LIN {X 0,Y 404.133,Z 474.142,A -85,B 0,C 180,E1 -11048.582,E2 -11048.582} C_VEL
LIN {X 0,Y 404.205,Z 474.132,A -85,B 0,C 180,E1 -11051.764,E2 -11051.764} C_VEL
LIN {X 0,Y 404.201,Z 474.136,A -85,B 0,C 180,E1 -11054.884,E2 -11054.884} C_VEL
LIN {X 0,Y 404.253,Z 474.125,A -85,B 0,C 180,E1 -11057.96,E2 -11057.96} C_VEL
LIN {X 0,Y 404.43,Z 474.108,A -85,B 0,C 180,E1 -11062.101,E2 -11062.101} C_VEL
LIN {X 0,Y 404.423,Z 474.111,A -85,B 0,C 180,E1 -11064.017,E2 -11064.017} C_VEL
LIN {X 0,Y 404.303,Z 474.258,A -85,B 0,C 180,E1 -11065.079,E2 -11065.079} C_VEL
LIN {X 0,Y 404.496,Z 475.213,A -85,B 0,C 180,E1 -11065.255,E2 -11065.255} C_VEL
LIN {X 0,Y 409.813,Z 489.68,A -85,B 0,C 180,E1 -11065.753,E2 -11065.753} C_VEL
LIN {X 0,Y 409.191,Z 554.574,A -85,B 0,C 180,E1 -11066.911,E2 -11066.911} C_VEL
LIN {X 0,Y 409.132,Z 567.718,A -85,B 0,C 180,E1 -11067.325,E2 -11067.325} C_VEL
LIN {X 0,Y 408.856,Z 581.109,A -85,B 0,C 180,E1 -11067.97,E2 -11067.97} C_VEL
LIN {X 0,Y 408.461,Z 593.219,A -85,B 0,C 180,E1 -11068.769,E2 -11068.769} C_VEL
LIN {X 0,Y 407.969,Z 603.324,A -85,B 0,C 180,E1 -11069.625,E2 -11069.625} C_VEL
LIN {X 0,Y 407.316,Z 613.938,A -85,B 0,C 180,E1 -11070.743,E2 -11070.743} C_VEL
LIN {X 0,Y 406.77,Z 623.415,A -85,B 0,C 180,E1 -11071.982,E2 -11071.982} C_VEL
LIN {X 0,Y 406.186,Z 631.224,A -85,B 0,C 180,E1 -11073.225,E2 -11073.225} C_VEL
LIN {X 0,Y 405.837,Z 635.869,A -85,B 0,C 180,E1 -11074.098,E2 -11074.098} C_VEL
LIN {X 0,Y 404.918,Z 639.248,A -85,B 0,C 180,E1 -11074.777,E2 -11074.777} C_VEL
LIN {X 0,Y 401.737,Z 644.43,A -85,B 0,C 180,E1 -11075.892,E2 -11075.892} C_VEL
LIN {X 0,Y 398.611,Z 648.964,A -85,B 0,C 180,E1 -11077.072,E2 -11077.072} C_VEL
LIN {X 0,Y 397.791,Z 651.292,A -85,B 0,C 180,E1 -11077.842,E2 -11077.842} C_VEL
LIN {X 0,Y 397.533,Z 654.48,A -85,B 0,C 180,E1 -11079.157,E2 -11079.157} C_VEL
LIN {X 0,Y 397.346,Z 656.459,A -85,B 0,C 180,E1 -11080.189,E2 -11080.189} C_VEL
LIN {X 0,Y 397.231,Z 658.018,A -85,B 0,C 180,E1 -11081.224,E2 -11081.224} C_VEL
LIN {X 0,Y 397.183,Z 659.113,A -85,B 0,C 180,E1 -11082.261,E2 -11082.261} C_VEL
LIN {X 0,Y 397.191,Z 659.81,A -85,B 0,C 180,E1 -11083.3,E2 -11083.3} C_VEL
LIN {X 0,Y 397.189,Z 660.13,A -85,B 0,C 180,E1 -11084.344,E2 -11084.344} C_VEL
LIN {X 0,Y 397.243,Z 660.03,A -85,B 0,C 180,E1 -11085.391,E2 -11085.391} C_VEL
LIN {X 0,Y 397.477,Z 658.759,A -85,B 0,C 180,E1 -11087.293,E2 -11087.293} C_VEL
LIN {X 0,Y 397.711,Z 657.198,A -85,B 0,C 180,E1 -11088.548,E2 -11088.548} C_VEL
LIN {X 0,Y 398.123,Z 654.276,A -85,B 0,C 180,E1 -11090.136,E2 -11090.136} C_VEL
LIN {X 0,Y 398.652,Z 650.226,A -85,B 0,C 180,E1 -11091.731,E2 -11091.731} C_VEL
LIN {X 0,Y 399.254,Z 644.972,A -85,B 0,C 180,E1 -11093.315,E2 -11093.315} C_VEL
LIN {X 0,Y 400.042,Z 638.106,A -85,B 0,C 180,E1 -11094.939,E2 -11094.939} C_VEL
LIN {X 0,Y 400.989,Z 629.888,A -85,B 0,C 180,E1 -11096.484,E2 -11096.484} C_VEL
LIN {X 0,Y 401.872,Z 620.477,A -85,B 0,C 180,E1 -11097.894,E2 -11097.894} C_VEL
LIN {X 0,Y 402.692,Z 610.549,A -85,B 0,C 180,E1 -11099.095,E2 -11099.095} C_VEL
LIN {X 0,Y 403.461,Z 600.695,A -85,B 0,C 180,E1 -11100.055,E2 -11100.055} C_VEL
LIN {X 0,Y 404.094,Z 589.275,A -85,B 0,C 180,E1 -11100.942,E2 -11100.942} C_VEL
LIN {X 0,Y 404.526,Z 577.358,A -85,B 0,C 180,E1 -11101.648,E2 -11101.648} C_VEL
LIN {X 0,Y 404.762,Z 564.049,A -85,B 0,C 180,E1 -11102.21,E2 -11102.21} C_VEL
LIN {X 0,Y 404.819,Z 549.962,A -85,B 0,C 180,E1 -11102.562,E2 -11102.562} C_VEL
LIN {X 0,Y 405.482,Z 494.287,A -85,B 0,C 180,E1 -11103.583,E2 -11103.583} C_VEL
LIN {X 0,Y 397.314,Z 475.91,A -85,B 0,C 180,E1 -11104.495,E2 -11104.495} C_VEL
LIN {X 0,Y 397.145,Z 475.073,A -85,B 0,C 180,E1 -11104.724,E2 -11104.724} C_VEL
LIN {X 0,Y 397.104,Z 475.022,A -85,B 0,C 180,E1 -11108.277,E2 -11108.277} C_VEL
LIN {X 0,Y 397.093,Z 475.024,A -85,B 0,C 180,E1 -11110.91,E2 -11110.91} C_VEL
LIN {X 0,Y 397.105,Z 475.019,A -85,B 0,C 180,E1 -11113.65,E2 -11113.65} C_VEL
LIN {X 0,Y 397.107,Z 475.021,A -85,B 0,C 180,E1 -11116.522,E2 -11116.522} C_VEL
LIN {X 0,Y 397.133,Z 475.196,A -85,B 0,C 180,E1 -11119.013,E2 -11119.013} C_VEL
LIN {X 0,Y 399.935,Z 487.895,A -85,B 0,C 180,E1 -11121.445,E2 -11121.445} C_VEL
LIN {X 0,Y 401.126,Z 495.291,A -85,B 0,C 180,E1 -11122.81,E2 -11122.81} C_VEL
LIN {X 0,Y 400.2,Z 516.124,A -85,B 0,C 180,E1 -11126.415,E2 -11126.415} C_VEL
LIN {X 0,Y 399.995,Z 522.02,A -85,B 0,C 180,E1 -11127.397,E2 -11127.397} C_VEL
LIN {X 0,Y 403.104,Z 541.761,A -85,B 0,C 180,E1 -11127.979,E2 -11127.979} C_VEL
LIN {X 0,Y 401.336,Z 632.644,A -85,B 0,C 180,E1 -11129.88,E2 -11129.88} C_VEL
LIN {X 0,Y 401.005,Z 645.03,A -85,B 0,C 180,E1 -11130.324,E2 -11130.324} C_VEL
LIN {X 0,Y 400.448,Z 657.146,A -85,B 0,C 180,E1 -11130.945,E2 -11130.945} C_VEL
LIN {X 0,Y 399.891,Z 669.821,A -85,B 0,C 180,E1 -11131.815,E2 -11131.815} C_VEL
LIN {X 0,Y 399.221,Z 680.557,A -85,B 0,C 180,E1 -11132.761,E2 -11132.761} C_VEL
LIN {X 0,Y 398.431,Z 692.076,A -85,B 0,C 180,E1 -11134.034,E2 -11134.034} C_VEL
LIN {X 0,Y 397.889,Z 700.606,A -85,B 0,C 180,E1 -11135.197,E2 -11135.197} C_VEL
LIN {X 0,Y 397.334,Z 708.675,A -85,B 0,C 180,E1 -11136.534,E2 -11136.534} C_VEL
LIN {X 0,Y 396.781,Z 716.618,A -85,B 0,C 180,E1 -11138.164,E2 -11138.164} C_VEL
LIN {X 0,Y 396.441,Z 722.686,A -85,B 0,C 180,E1 -11139.733,E2 -11139.733} C_VEL
LIN {X 0,Y 396.136,Z 727.578,A -85,B 0,C 180,E1 -11141.377,E2 -11141.377} C_VEL
LIN {X 0,Y 396.042,Z 730.058,A -85,B 0,C 180,E1 -11142.442,E2 -11142.442} C_VEL
LIN {X 0,Y 395.913,Z 732.043,A -85,B 0,C 180,E1 -11143.5,E2 -11143.5} C_VEL
LIN {X 0,Y 395.806,Z 733.503,A -85,B 0,C 180,E1 -11144.554,E2 -11144.554} C_VEL
LIN {X 0,Y 395.753,Z 734.538,A -85,B 0,C 180,E1 -11145.605,E2 -11145.605} C_VEL
LIN {X 0,Y 395.865,Z 735.231,A -85,B 0,C 180,E1 -11147.544,E2 -11147.544} C_VEL
LIN {X 0,Y 395.892,Z 734.913,A -85,B 0,C 180,E1 -11148.74,E2 -11148.74} C_VEL
LIN {X 0,Y 395.902,Z 734.17,A -85,B 0,C 180,E1 -11149.775,E2 -11149.775} C_VEL
LIN {X 0,Y 396.034,Z 732.96,A -85,B 0,C 180,E1 -11150.81,E2 -11150.81} C_VEL
LIN {X 0,Y 396.277,Z 730.336,A -85,B 0,C 180,E1 -11152.357,E2 -11152.357} C_VEL
LIN {X 0,Y 396.521,Z 726.682,A -85,B 0,C 180,E1 -11153.896,E2 -11153.896} C_VEL
LIN {X 0,Y 396.894,Z 721.882,A -85,B 0,C 180,E1 -11155.43,E2 -11155.43} C_VEL
LIN {X 0,Y 397.41,Z 715.803,A -85,B 0,C 180,E1 -11156.959,E2 -11156.959} C_VEL
LIN {X 0,Y 398.122,Z 708.162,A -85,B 0,C 180,E1 -11158.483,E2 -11158.483} C_VEL
LIN {X 0,Y 399.009,Z 698.649,A -85,B 0,C 180,E1 -11160,E2 -11160} C_VEL
LIN {X 0,Y 399.831,Z 688.759,A -85,B 0,C 180,E1 -11161.259,E2 -11161.259} C_VEL
LIN {X 0,Y 400.716,Z 677.71,A -85,B 0,C 180,E1 -11162.388,E2 -11162.388} C_VEL
LIN {X 0,Y 401.413,Z 666.543,A -85,B 0,C 180,E1 -11163.301,E2 -11163.301} C_VEL
LIN {X 0,Y 402.197,Z 653.515,A -85,B 0,C 180,E1 -11164.108,E2 -11164.108} C_VEL
LIN {X 0,Y 402.666,Z 640.568,A -85,B 0,C 180,E1 -11164.692,E2 -11164.692} C_VEL
LIN {X 0,Y 403.089,Z 626.256,A -85,B 0,C 180,E1 -11165.096,E2 -11165.096} C_VEL
LIN {X 0,Y 405.254,Z 541.083,A -85,B 0,C 180,E1 -11166.99,E2 -11166.99} C_VEL
LIN {X 0,Y 402.058,Z 526.063,A -85,B 0,C 180,E1 -11167.597,E2 -11167.597} C_VEL
LIN {X 0,Y 401.812,Z 524.403,A -85,B 0,C 180,E1 -11167.728,E2 -11167.728} C_VEL
LIN {X 0,Y 402.819,Z 502.886,A -85,B 0,C 180,E1 -11171.411,E2 -11171.411} C_VEL
LIN {X 0,Y 403.071,Z 499.016,A -85,B 0,C 180,E1 -11172.078,E2 -11172.078} C_VEL
LIN {X 0,Y 401.479,Z 490.655,A -85,B 0,C 180,E1 -11173.67,E2 -11173.67} C_VEL
LIN {X 0,Y 398.591,Z 479.718,A -85,B 0,C 180,E1 -11175.861,E2 -11175.861} C_VEL
LIN {X 0,Y 397.195,Z 475.127,A -85,B 0,C 180,E1 -11176.877,E2 -11176.877} C_VEL
LIN {X 0,Y 397.148,Z 475.016,A -85,B 0,C 180,E1 -11180.295,E2 -11180.295} C_VEL
LIN {X 0,Y 397.134,Z 475.017,A -85,B 0,C 180,E1 -11184.019,E2 -11184.019} C_VEL
LIN {X 0,Y 397.203,Z 475.009,A -85,B 0,C 180,E1 -11187.39,E2 -11187.39} C_VEL
LIN {X 0,Y 397.088,Z 475.024,A -85,B 0,C 180,E1 -11190.882,E2 -11190.882} C_VEL
LIN {X 0,Y 397.134,Z 475.016,A -85,B 0,C 180,E1 -11194.493,E2 -11194.493} C_VEL
LIN {X 0,Y 397.11,Z 475.017,A -85,B 0,C 180,E1 -11198.275,E2 -11198.275} C_VEL
LIN {X 0,Y 397.097,Z 475.023,A -85,B 0,C 180,E1 -11200.908,E2 -11200.908} C_VEL
LIN {X 0,Y 397.109,Z 475.019,A -85,B 0,C 180,E1 -11203.648,E2 -11203.648} C_VEL
LIN {X 0,Y 397.11,Z 475.018,A -85,B 0,C 180,E1 -11206.52,E2 -11206.52} C_VEL
LIN {X 0,Y 397.12,Z 475.008,A -85,B 0,C 180,E1 -11210.422,E2 -11210.422} C_VEL
LIN {X 0,Y 397.104,Z 475.007,A -85,B 0,C 180,E1 -11213.004,E2 -11213.004} C_VEL
LIN {X 0,Y 397.146,Z 475.218,A -85,B 0,C 180,E1 -11215.91,E2 -11215.91} C_VEL
LIN {X 0,Y 400.382,Z 487.87,A -85,B 0,C 180,E1 -11218.488,E2 -11218.488} C_VEL
LIN {X 0,Y 402.986,Z 499.886,A -85,B 0,C 180,E1 -11220.769,E2 -11220.769} C_VEL
LIN {X 0,Y 402.926,Z 503.223,A -85,B 0,C 180,E1 -11221.335,E2 -11221.335} C_VEL
LIN {X 0,Y 401.063,Z 524.8,A -85,B 0,C 180,E1 -11224.851,E2 -11224.851} C_VEL
LIN {X 0,Y 399.235,Z 550.114,A -85,B 0,C 180,E1 -11228.907,E2 -11228.907} C_VEL
LIN {X 0,Y 399.204,Z 552.057,A -85,B 0,C 180,E1 -11229.132,E2 -11229.132} C_VEL
LIN {X 0,Y 400.616,Z 562.417,A -85,B 0,C 180,E1 -11229.554,E2 -11229.554} C_VEL
LIN {X 0,Y 403.001,Z 585.438,A -85,B 0,C 180,E1 -11230.266,E2 -11230.266} C_VEL
LIN {X 0,Y 403.893,Z 597.547,A -85,B 0,C 180,E1 -11230.544,E2 -11230.544} C_VEL
LIN {X 0,Y 402.92,Z 664.118,A -85,B 0,C 180,E1 -11231.766,E2 -11231.766} C_VEL
LIN {X 0,Y 402.288,Z 677.425,A -85,B 0,C 180,E1 -11232.197,E2 -11232.197} C_VEL
LIN {X 0,Y 401.369,Z 690.214,A -85,B 0,C 180,E1 -11232.812,E2 -11232.812} C_VEL
LIN {X 0,Y 399.991,Z 709.915,A -85,B 0,C 180,E1 -11234.064,E2 -11234.064} C_VEL
LIN {X 0,Y 399.197,Z 720.793,A -85,B 0,C 180,E1 -11234.947,E2 -11234.947} C_VEL
LIN {X 0,Y 398.466,Z 730.713,A -85,B 0,C 180,E1 -11235.948,E2 -11235.948} C_VEL
LIN {X 0,Y 397.619,Z 741.025,A -85,B 0,C 180,E1 -11237.234,E2 -11237.234} C_VEL
LIN {X 0,Y 397.105,Z 749.384,A -85,B 0,C 180,E1 -11238.514,E2 -11238.514} C_VEL
LIN {X 0,Y 396.569,Z 757.583,A -85,B 0,C 180,E1 -11240.048,E2 -11240.048} C_VEL
LIN {X 0,Y 396.182,Z 765.089,A -85,B 0,C 180,E1 -11241.84,E2 -11241.84} C_VEL
LIN {X 0,Y 395.994,Z 770.249,A -85,B 0,C 180,E1 -11243.425,E2 -11243.425} C_VEL
LIN {X 0,Y 395.987,Z 773.916,A -85,B 0,C 180,E1 -11244.907,E2 -11244.907} C_VEL
LIN {X 0,Y 395.92,Z 775.85,A -85,B 0,C 180,E1 -11245.927,E2 -11245.927} C_VEL
LIN {X 0,Y 395.972,Z 777.314,A -85,B 0,C 180,E1 -11246.946,E2 -11246.946} C_VEL
LIN {X 0,Y 396.014,Z 778.36,A -85,B 0,C 180,E1 -11247.964,E2 -11247.964} C_VEL
LIN {X 0,Y 395.992,Z 778.965,A -85,B 0,C 180,E1 -11248.981,E2 -11248.981} C_VEL
LIN {X 0,Y 396.085,Z 779.104,A -85,B 0,C 180,E1 -11249.998,E2 -11249.998} C_VEL
LIN {X 0,Y 396.014,Z 778.816,A -85,B 0,C 180,E1 -11251.015,E2 -11251.015} C_VEL
LIN {X 0,Y 396.013,Z 778.114,A -85,B 0,C 180,E1 -11252.032,E2 -11252.032} C_VEL
LIN {X 0,Y 396.018,Z 776.927,A -85,B 0,C 180,E1 -11253.05,E2 -11253.05} C_VEL
LIN {X 0,Y 395.971,Z 774.309,A -85,B 0,C 180,E1 -11254.579,E2 -11254.579} C_VEL
LIN {X 0,Y 395.971,Z 770.015,A -85,B 0,C 180,E1 -11256.313,E2 -11256.313} C_VEL
LIN {X 0,Y 396.099,Z 765.675,A -85,B 0,C 180,E1 -11257.645,E2 -11257.645} C_VEL
LIN {X 0,Y 396.328,Z 759.409,A -85,B 0,C 180,E1 -11259.182,E2 -11259.182} C_VEL
LIN {X 0,Y 396.698,Z 751.537,A -85,B 0,C 180,E1 -11260.719,E2 -11260.719} C_VEL
LIN {X 0,Y 397.179,Z 743.415,A -85,B 0,C 180,E1 -11261.998,E2 -11261.998} C_VEL
LIN {X 0,Y 397.828,Z 734.585,A -85,B 0,C 180,E1 -11263.145,E2 -11263.145} C_VEL
LIN {X 0,Y 398.362,Z 723.74,A -85,B 0,C 180,E1 -11264.298,E2 -11264.298} C_VEL
LIN {X 0,Y 399.039,Z 713.221,A -85,B 0,C 180,E1 -11265.186,E2 -11265.186} C_VEL
LIN {X 0,Y 399.761,Z 700.61,A -85,B 0,C 180,E1 -11266.007,E2 -11266.007} C_VEL
LIN {X 0,Y 400.839,Z 683.335,A -85,B 0,C 180,E1 -11266.945,E2 -11266.945} C_VEL
LIN {X 0,Y 401.414,Z 670.298,A -85,B 0,C 180,E1 -11267.445,E2 -11267.445} C_VEL
LIN {X 0,Y 401.724,Z 654.557,A -85,B 0,C 180,E1 -11267.793,E2 -11267.793} C_VEL
LIN {X 0,Y 402.305,Z 593.458,A -85,B 0,C 180,E1 -11268.885,E2 -11268.885} C_VEL
LIN {X 0,Y 398.442,Z 555.652,A -85,B 0,C 180,E1 -11269.746,E2 -11269.746} C_VEL
LIN {X 0,Y 398.417,Z 554.31,A -85,B 0,C 180,E1 -11269.848,E2 -11269.848} C_VEL
LIN {X 0,Y 399.688,Z 532.021,A -85,B 0,C 180,E1 -11273.303,E2 -11273.303} C_VEL
LIN {X 0,Y 401.324,Z 507.919,A -85,B 0,C 180,E1 -11277.083,E2 -11277.083} C_VEL
LIN {X 0,Y 401.936,Z 497.094,A -85,B 0,C 180,E1 -11278.805,E2 -11278.805} C_VEL
LIN {X 0,Y 397.969,Z 478.817,A -85,B 0,C 180,E1 -11282.041,E2 -11282.041} C_VEL
LIN {X 0,Y 397.143,Z 475.144,A -85,B 0,C 180,E1 -11282.738,E2 -11282.738} C_VEL
LIN {X 0,Y 397.1,Z 475.022,A -85,B 0,C 180,E1 -11285.733,E2 -11285.733} C_VEL
LIN {X 0,Y 397.084,Z 475.019,A -85,B 0,C 180,E1 -11288.852,E2 -11288.852} C_VEL
LIN {X 0,Y 397.048,Z 475.029,A -85,B 0,C 180,E1 -11292.267,E2 -11292.267} C_VEL
LIN {X 0,Y 397.077,Z 475.019,A -85,B 0,C 180,E1 -11295.067,E2 -11295.067} C_VEL
LIN {X 0,Y 397.05,Z 475.027,A -85,B 0,C 180,E1 -11298.021,E2 -11298.021} C_VEL
LIN {X 0,Y 397.084,Z 475.018,A -85,B 0,C 180,E1 -11301.144,E2 -11301.144} C_VEL
LIN {X 0,Y 397.108,Z 475.02,A -85,B 0,C 180,E1 -11304.495,E2 -11304.495} C_VEL
LIN {X 0,Y 397.067,Z 475.023,A -85,B 0,C 180,E1 -11307.927,E2 -11307.927} C_VEL
LIN {X 0,Y 397.11,Z 475.015,A -85,B 0,C 180,E1 -11311.455,E2 -11311.455} C_VEL
LIN {X 0,Y 397.139,Z 475.017,A -85,B 0,C 180,E1 -11314.487,E2 -11314.487} C_VEL
LIN {X 0,Y 397.096,Z 475.022,A -85,B 0,C 180,E1 -11318.181,E2 -11318.181} C_VEL
LIN {X 0,Y 397.149,Z 475.01,A -85,B 0,C 180,E1 -11321.426,E2 -11321.426} C_VEL
LIN {X 0,Y 397.165,Z 475.013,A -85,B 0,C 180,E1 -11324.607,E2 -11324.607} C_VEL
LIN {X 0,Y 397.207,Z 475.004,A -85,B 0,C 180,E1 -11327.741,E2 -11327.741} C_VEL
LIN {X 0,Y 397.381,Z 474.984,A -85,B 0,C 180,E1 -11332.041,E2 -11332.041} C_VEL
LIN {X 0,Y 397.238,Z 475.002,A -85,B 0,C 180,E1 -11334.925,E2 -11334.925} C_VEL
LIN {X 0,Y 397.435,Z 474.976,A -85,B 0,C 180,E1 -11337.973,E2 -11337.973} C_VEL
LIN {X 0,Y 397.566,Z 474.96,A -85,B 0,C 180,E1 -11340,E2 -11340} C_VEL
LIN {X 0,Y 397.366,Z 474.985,A -85,B 0,C 180,E1 -11343.041,E2 -11343.041} C_VEL
LIN {X 0,Y 397.348,Z 474.987,A -85,B 0,C 180,E1 -11347.112,E2 -11347.112} C_VEL
LIN {X 0,Y 397.205,Z 475.006,A -85,B 0,C 180,E1 -11350.191,E2 -11350.191} C_VEL
LIN {X 0,Y 397.212,Z 475.003,A -85,B 0,C 180,E1 -11353.321,E2 -11353.321} C_VEL
LIN {X 0,Y 397.167,Z 475.01,A -85,B 0,C 180,E1 -11357.155,E2 -11357.155} C_VEL
LIN {X 0,Y 397.088,Z 475.025,A -85,B 0,C 180,E1 -11360.73,E2 -11360.73} C_VEL
LIN {X 0,Y 397.119,Z 475.014,A -85,B 0,C 180,E1 -11364.019,E2 -11364.019} C_VEL
LIN {X 0,Y 397.181,Z 475.007,A -85,B 0,C 180,E1 -11367.391,E2 -11367.391} C_VEL
LIN {X 0,Y 397.066,Z 475.027,A -85,B 0,C 180,E1 -11370.883,E2 -11370.883} C_VEL
LIN {X 0,Y 397.113,Z 475.018,A -85,B 0,C 180,E1 -11374.494,E2 -11374.494} C_VEL
LIN {X 0,Y 397.092,Z 475.019,A -85,B 0,C 180,E1 -11378.276,E2 -11378.276} C_VEL
LIN {X 0,Y 397.077,Z 475.026,A -85,B 0,C 180,E1 -11380.91,E2 -11380.91} C_VEL
LIN {X 0,Y 397.094,Z 475.017,A -85,B 0,C 180,E1 -11383.649,E2 -11383.649} C_VEL
LIN {X 0,Y 397.149,Z 475.013,A -85,B 0,C 180,E1 -11386.513,E2 -11386.513} C_VEL
LIN {X 0,Y 397.114,Z 475.016,A -85,B 0,C 180,E1 -11389.552,E2 -11389.552} C_VEL
LIN {X 0,Y 397.113,Z 475.02,A -85,B 0,C 180,E1 -11392.787,E2 -11392.787} C_VEL
LIN {X 0,Y 397.109,Z 475.016,A -85,B 0,C 180,E1 -11396.284,E2 -11396.284} C_VEL
LIN {X 0,Y 397.097,Z 475.017,A -85,B 0,C 180,E1 -11400.137,E2 -11400.137} C_VEL
LIN {X 0,Y 397.187,Z 475.008,A -85,B 0,C 180,E1 -11402.611,E2 -11402.611} C_VEL
LIN {X 0,Y 397.126,Z 475.013,A -85,B 0,C 180,E1 -11405.983,E2 -11405.983} C_VEL
LIN {X 0,Y 397.132,Z 475.013,A -85,B 0,C 180,E1 -11409.706,E2 -11409.706} C_VEL
LIN {X 0,Y 397.176,Z 475.011,A -85,B 0,C 180,E1 -11412.846,E2 -11412.846} C_VEL
LIN {X 0,Y 397.224,Z 475.003,A -85,B 0,C 180,E1 -11416.704,E2 -11416.704} C_VEL
LIN {X 0,Y 397.215,Z 475.007,A -85,B 0,C 180,E1 -11419.811,E2 -11419.811} C_VEL
LIN {X 0,Y 397.362,Z 474.988,A -85,B 0,C 180,E1 -11422.89,E2 -11422.89} C_VEL
LIN {X 0,Y 397.274,Z 475.174,A -85,B 0,C 180,E1 -11424.8,E2 -11424.8} C_VEL
LIN {X 0,Y 397.434,Z 476.035,A -85,B 0,C 180,E1 -11424.957,E2 -11424.957} C_VEL
LIN {X 0,Y 402.904,Z 491.025,A -85,B 0,C 180,E1 -11425.492,E2 -11425.492} C_VEL
LIN {X 0,Y 402.371,Z 556.242,A -85,B 0,C 180,E1 -11426.68,E2 -11426.68} C_VEL
LIN {X 0,Y 402.262,Z 569.599,A -85,B 0,C 180,E1 -11427.123,E2 -11427.123} C_VEL
LIN {X 0,Y 401.992,Z 582.198,A -85,B 0,C 180,E1 -11427.747,E2 -11427.747} C_VEL
LIN {X 0,Y 401.614,Z 593.455,A -85,B 0,C 180,E1 -11428.498,E2 -11428.498} C_VEL
LIN {X 0,Y 401.072,Z 604.477,A -85,B 0,C 180,E1 -11429.442,E2 -11429.442} C_VEL
LIN {X 0,Y 400.362,Z 615.489,A -85,B 0,C 180,E1 -11430.63,E2 -11430.63} C_VEL
LIN {X 0,Y 399.883,Z 623.984,A -85,B 0,C 180,E1 -11431.764,E2 -11431.764} C_VEL
LIN {X 0,Y 399.269,Z 631.862,A -85,B 0,C 180,E1 -11433.029,E2 -11433.029} C_VEL
LIN {X 0,Y 398.681,Z 639.577,A -85,B 0,C 180,E1 -11434.552,E2 -11434.552} C_VEL
LIN {X 0,Y 398.214,Z 645.749,A -85,B 0,C 180,E1 -11436.08,E2 -11436.08} C_VEL
LIN {X 0,Y 397.791,Z 651.292,A -85,B 0,C 180,E1 -11437.842,E2 -11437.842} C_VEL
LIN {X 0,Y 396.97,Z 653.417,A -85,B 0,C 180,E1 -11438.629,E2 -11438.629} C_VEL
LIN {X 0,Y 393.875,Z 656.494,A -85,B 0,C 180,E1 -11439.919,E2 -11439.919} C_VEL
LIN {X 0,Y 391.324,Z 658.509,A -85,B 0,C 180,E1 -11440.982,E2 -11440.982} C_VEL
LIN {X 0,Y 390.234,Z 659.652,A -85,B 0,C 180,E1 -11441.819,E2 -11441.819} C_VEL
LIN {X 0,Y 390.147,Z 659.892,A -85,B 0,C 180,E1 -11442.105,E2 -11442.105} C_VEL
LIN {X 0,Y 390.166,Z 660.9,A -85,B 0,C 180,E1 -11443.544,E2 -11443.544} C_VEL
LIN {X 0,Y 390.166,Z 661.14,A -85,B 0,C 180,E1 -11444.608,E2 -11444.608} C_VEL
LIN {X 0,Y 390.253,Z 660.934,A -85,B 0,C 180,E1 -11445.674,E2 -11445.674} C_VEL
LIN {X 0,Y 390.487,Z 659.688,A -85,B 0,C 180,E1 -11447.467,E2 -11447.467} C_VEL
LIN {X 0,Y 390.768,Z 657.858,A -85,B 0,C 180,E1 -11448.89,E2 -11448.89} C_VEL
LIN {X 0,Y 391.222,Z 654.876,A -85,B 0,C 180,E1 -11450.474,E2 -11450.474} C_VEL
LIN {X 0,Y 391.827,Z 650.601,A -85,B 0,C 180,E1 -11452.129,E2 -11452.129} C_VEL
LIN {X 0,Y 392.46,Z 645.466,A -85,B 0,C 180,E1 -11453.668,E2 -11453.668} C_VEL
LIN {X 0,Y 393.381,Z 638.154,A -85,B 0,C 180,E1 -11455.391,E2 -11455.391} C_VEL
LIN {X 0,Y 394.256,Z 630.587,A -85,B 0,C 180,E1 -11456.809,E2 -11456.809} C_VEL
LIN {X 0,Y 395.212,Z 620.96,A -85,B 0,C 180,E1 -11458.261,E2 -11458.261} C_VEL
LIN {X 0,Y 396.059,Z 611.137,A -85,B 0,C 180,E1 -11459.458,E2 -11459.458} C_VEL
LIN {X 0,Y 396.907,Z 600.915,A -85,B 0,C 180,E1 -11460.457,E2 -11460.457} C_VEL
LIN {X 0,Y 397.578,Z 589.209,A -85,B 0,C 180,E1 -11461.359,E2 -11461.359} C_VEL
LIN {X 0,Y 398.043,Z 576.36,A -85,B 0,C 180,E1 -11462.107,E2 -11462.107} C_VEL
LIN {X 0,Y 398.233,Z 564.269,A -85,B 0,C 180,E1 -11462.604,E2 -11462.604} C_VEL
LIN {X 0,Y 398.269,Z 549.837,A -85,B 0,C 180,E1 -11462.958,E2 -11462.958} C_VEL
LIN {X 0,Y 399.017,Z 496.122,A -85,B 0,C 180,E1 -11463.956,E2 -11463.956} C_VEL
LIN {X 0,Y 390.342,Z 476.97,A -85,B 0,C 180,E1 -11464.937,E2 -11464.937} C_VEL
LIN {X 0,Y 390.134,Z 476.02,A -85,B 0,C 180,E1 -11465.134,E2 -11465.134} C_VEL
LIN {X 0,Y 390.071,Z 475.89,A -85,B 0,C 180,E1 -11469.219,E2 -11469.219} C_VEL
LIN {X 0,Y 390.046,Z 475.892,A -85,B 0,C 180,E1 -11472.375,E2 -11472.375} C_VEL
LIN {X 0,Y 390.049,Z 475.901,A -85,B 0,C 180,E1 -11475.356,E2 -11475.356} C_VEL
LIN {X 0,Y 390.104,Z 476.111,A -85,B 0,C 180,E1 -11478.743,E2 -11478.743} C_VEL
LIN {X 0,Y 393.147,Z 490.003,A -85,B 0,C 180,E1 -11481.429,E2 -11481.429} C_VEL
LIN {X 0,Y 394.23,Z 496.767,A -85,B 0,C 180,E1 -11482.691,E2 -11482.691} C_VEL
LIN {X 0,Y 393.279,Z 517.823,A -85,B 0,C 180,E1 -11486.36,E2 -11486.36} C_VEL
LIN {X 0,Y 393.127,Z 522.4,A -85,B 0,C 180,E1 -11487.112,E2 -11487.112} C_VEL
LIN {X 0,Y 396.267,Z 542.631,A -85,B 0,C 180,E1 -11487.716,E2 -11487.716} C_VEL
LIN {X 0,Y 394.465,Z 632.37,A -85,B 0,C 180,E1 -11489.633,E2 -11489.633} C_VEL
LIN {X 0,Y 394.077,Z 645.723,A -85,B 0,C 180,E1 -11490.117,E2 -11490.117} C_VEL
LIN {X 0,Y 393.495,Z 658.628,A -85,B 0,C 180,E1 -11490.804,E2 -11490.804} C_VEL
LIN {X 0,Y 392.882,Z 671.217,A -85,B 0,C 180,E1 -11491.704,E2 -11491.704} C_VEL
LIN {X 0,Y 392.096,Z 683.083,A -85,B 0,C 180,E1 -11492.802,E2 -11492.802} C_VEL
LIN {X 0,Y 391.45,Z 692.306,A -85,B 0,C 180,E1 -11493.859,E2 -11493.859} C_VEL
LIN {X 0,Y 390.899,Z 700.635,A -85,B 0,C 180,E1 -11495.007,E2 -11495.007} C_VEL
LIN {X 0,Y 390.311,Z 708.872,A -85,B 0,C 180,E1 -11496.382,E2 -11496.382} C_VEL
LIN {X 0,Y 389.743,Z 716.8,A -85,B 0,C 180,E1 -11498.027,E2 -11498.027} C_VEL
LIN {X 0,Y 389.418,Z 722.111,A -85,B 0,C 180,E1 -11499.396,E2 -11499.396} C_VEL
LIN {X 0,Y 389.119,Z 727.167,A -85,B 0,C 180,E1 -11501.029,E2 -11501.029} C_VEL
LIN {X 0,Y 388.928,Z 730.941,A -85,B 0,C 180,E1 -11502.653,E2 -11502.653} C_VEL
LIN {X 0,Y 388.746,Z 733.557,A -85,B 0,C 180,E1 -11504.266,E2 -11504.266} C_VEL
LIN {X 0,Y 388.666,Z 734.691,A -85,B 0,C 180,E1 -11505.336,E2 -11505.336} C_VEL
LIN {X 0,Y 388.681,Z 735.399,A -85,B 0,C 180,E1 -11506.405,E2 -11506.405} C_VEL
LIN {X 0,Y 388.777,Z 735.659,A -85,B 0,C 180,E1 -11507.472,E2 -11507.472} C_VEL
LIN {X 0,Y 388.798,Z 735.452,A -85,B 0,C 180,E1 -11508.531,E2 -11508.531} C_VEL
LIN {X 0,Y 388.811,Z 734.839,A -85,B 0,C 180,E1 -11509.587,E2 -11509.587} C_VEL
LIN {X 0,Y 388.927,Z 733.79,A -85,B 0,C 180,E1 -11510.641,E2 -11510.641} C_VEL
LIN {X 0,Y 389.106,Z 732.263,A -85,B 0,C 180,E1 -11511.692,E2 -11511.692} C_VEL
LIN {X 0,Y 389.357,Z 729.501,A -85,B 0,C 180,E1 -11513.114,E2 -11513.114} C_VEL
LIN {X 0,Y 389.688,Z 724.963,A -85,B 0,C 180,E1 -11514.827,E2 -11514.827} C_VEL
LIN {X 0,Y 390.197,Z 719.549,A -85,B 0,C 180,E1 -11516.386,E2 -11516.386} C_VEL
LIN {X 0,Y 390.821,Z 712.766,A -85,B 0,C 180,E1 -11517.939,E2 -11517.939} C_VEL
LIN {X 0,Y 391.694,Z 704.236,A -85,B 0,C 180,E1 -11519.486,E2 -11519.486} C_VEL
LIN {X 0,Y 392.493,Z 695.586,A -85,B 0,C 180,E1 -11520.77,E2 -11520.77} C_VEL
LIN {X 0,Y 393.34,Z 686.106,A -85,B 0,C 180,E1 -11521.92,E2 -11521.92} C_VEL
LIN {X 0,Y 394.298,Z 674.251,A -85,B 0,C 180,E1 -11523.066,E2 -11523.066} C_VEL
LIN {X 0,Y 395.073,Z 662.419,A -85,B 0,C 180,E1 -11523.963,E2 -11523.963} C_VEL
LIN {X 0,Y 395.797,Z 649.128,A -85,B 0,C 180,E1 -11524.711,E2 -11524.711} C_VEL
LIN {X 0,Y 396.273,Z 636.449,A -85,B 0,C 180,E1 -11525.215,E2 -11525.215} C_VEL
LIN {X 0,Y 397.161,Z 600.168,A -85,B 0,C 180,E1 -11526.063,E2 -11526.063} C_VEL
LIN {X 0,Y 398.807,Z 542.016,A -85,B 0,C 180,E1 -11527.421,E2 -11527.421} C_VEL
LIN {X 0,Y 395.372,Z 525.895,A -85,B 0,C 180,E1 -11528.112,E2 -11528.112} C_VEL
LIN {X 0,Y 395.235,Z 525.113,A -85,B 0,C 180,E1 -11528.179,E2 -11528.179} C_VEL
LIN {X 0,Y 396.335,Z 503.605,A -85,B 0,C 180,E1 -11531.893,E2 -11531.893} C_VEL
LIN {X 0,Y 396.328,Z 499.729,A -85,B 0,C 180,E1 -11532.567,E2 -11532.567} C_VEL
LIN {X 0,Y 394.288,Z 490.321,A -85,B 0,C 180,E1 -11534.451,E2 -11534.451} C_VEL
LIN {X 0,Y 391.239,Z 479.486,A -85,B 0,C 180,E1 -11536.704,E2 -11536.704} C_VEL
LIN {X 0,Y 390.138,Z 476.002,A -85,B 0,C 180,E1 -11537.536,E2 -11537.536} C_VEL
LIN {X 0,Y 390.064,Z 475.898,A -85,B 0,C 180,E1 -11541.122,E2 -11541.122} C_VEL
LIN {X 0,Y 390.084,Z 475.897,A -85,B 0,C 180,E1 -11544.481,E2 -11544.481} C_VEL
LIN {X 0,Y 390.127,Z 475.889,A -85,B 0,C 180,E1 -11547.93,E2 -11547.93} C_VEL
LIN {X 0,Y 390.032,Z 475.9,A -85,B 0,C 180,E1 -11551.504,E2 -11551.504} C_VEL
LIN {X 0,Y 390.094,Z 475.893,A -85,B 0,C 180,E1 -11555.206,E2 -11555.206} C_VEL
LIN {X 0,Y 390.077,Z 475.896,A -85,B 0,C 180,E1 -11559.217,E2 -11559.217} C_VEL
LIN {X 0,Y 390.051,Z 475.897,A -85,B 0,C 180,E1 -11562.373,E2 -11562.373} C_VEL
LIN {X 0,Y 390.053,Z 475.898,A -85,B 0,C 180,E1 -11565.354,E2 -11565.354} C_VEL
LIN {X 0,Y 390.039,Z 475.899,A -85,B 0,C 180,E1 -11568.186,E2 -11568.186} C_VEL
LIN {X 0,Y 390.094,Z 475.874,A -85,B 0,C 180,E1 -11570.906,E2 -11570.906} C_VEL
LIN {X 0,Y 390.078,Z 475.884,A -85,B 0,C 180,E1 -11574.791,E2 -11574.791} C_VEL
LIN {X 0,Y 390.123,Z 476.129,A -85,B 0,C 180,E1 -11575.474,E2 -11575.474} C_VEL
LIN {X 0,Y 393.478,Z 489.209,A -85,B 0,C 180,E1 -11578.202,E2 -11578.202} C_VEL
LIN {X 0,Y 396.218,Z 501.721,A -85,B 0,C 180,E1 -11580.631,E2 -11580.631} C_VEL
LIN {X 0,Y 395.494,Z 510.964,A -85,B 0,C 180,E1 -11582.193,E2 -11582.193} C_VEL
LIN {X 0,Y 393.647,Z 532.503,A -85,B 0,C 180,E1 -11585.754,E2 -11585.754} C_VEL
LIN {X 0,Y 392.37,Z 549.363,A -85,B 0,C 180,E1 -11588.482,E2 -11588.482} C_VEL
LIN {X 0,Y 393.027,Z 555.201,A -85,B 0,C 180,E1 -11588.813,E2 -11588.813} C_VEL
LIN {X 0,Y 395.193,Z 571.979,A -85,B 0,C 180,E1 -11589.419,E2 -11589.419} C_VEL
LIN {X 0,Y 397.032,Z 593.132,A -85,B 0,C 180,E1 -11590.069,E2 -11590.069} C_VEL
LIN {X 0,Y 397.231,Z 600.364,A -85,B 0,C 180,E1 -11590.221,E2 -11590.221} C_VEL
LIN {X 0,Y 396.264,Z 663.763,A -85,B 0,C 180,E1 -11591.415,E2 -11591.415} C_VEL
LIN {X 0,Y 395.569,Z 676.847,A -85,B 0,C 180,E1 -11591.85,E2 -11591.85} C_VEL
LIN {X 0,Y 394.602,Z 690.077,A -85,B 0,C 180,E1 -11592.508,E2 -11592.508} C_VEL
LIN {X 0,Y 393.43,Z 706.717,A -85,B 0,C 180,E1 -11593.524,E2 -11593.524} C_VEL
LIN {X 0,Y 392.475,Z 719.467,A -85,B 0,C 180,E1 -11594.55,E2 -11594.55} C_VEL
LIN {X 0,Y 391.602,Z 729.995,A -85,B 0,C 180,E1 -11595.617,E2 -11595.617} C_VEL
LIN {X 0,Y 390.852,Z 739.091,A -85,B 0,C 180,E1 -11596.745,E2 -11596.745} C_VEL
LIN {X 0,Y 390.266,Z 747.701,A -85,B 0,C 180,E1 -11598.046,E2 -11598.046} C_VEL
LIN {X 0,Y 389.596,Z 756.141,A -85,B 0,C 180,E1 -11599.606,E2 -11599.606} C_VEL
LIN {X 0,Y 389.224,Z 762.93,A -85,B 0,C 180,E1 -11601.17,E2 -11601.17} C_VEL
LIN {X 0,Y 388.957,Z 768.294,A -85,B 0,C 180,E1 -11602.732,E2 -11602.732} C_VEL
LIN {X 0,Y 388.854,Z 771.92,A -85,B 0,C 180,E1 -11604.064,E2 -11604.064} C_VEL
LIN {X 0,Y 388.839,Z 775.501,A -85,B 0,C 180,E1 -11605.852,E2 -11605.852} C_VEL
LIN {X 0,Y 388.871,Z 776.957,A -85,B 0,C 180,E1 -11606.89,E2 -11606.89} C_VEL
LIN {X 0,Y 388.94,Z 777.992,A -85,B 0,C 180,E1 -11607.927,E2 -11607.927} C_VEL
LIN {X 0,Y 388.914,Z 778.565,A -85,B 0,C 180,E1 -11608.963,E2 -11608.963} C_VEL
LIN {X 0,Y 388.998,Z 778.688,A -85,B 0,C 180,E1 -11609.998,E2 -11609.998} C_VEL
LIN {X 0,Y 388.933,Z 778.385,A -85,B 0,C 180,E1 -11611.034,E2 -11611.034} C_VEL
LIN {X 0,Y 388.941,Z 777.654,A -85,B 0,C 180,E1 -11612.069,E2 -11612.069} C_VEL
LIN {X 0,Y 388.917,Z 776.435,A -85,B 0,C 180,E1 -11613.106,E2 -11613.106} C_VEL
LIN {X 0,Y 388.903,Z 773.774,A -85,B 0,C 180,E1 -11614.663,E2 -11614.663} C_VEL
LIN {X 0,Y 388.891,Z 769.789,A -85,B 0,C 180,E1 -11616.3,E2 -11616.3} C_VEL
LIN {X 0,Y 389.04,Z 765.029,A -85,B 0,C 180,E1 -11617.785,E2 -11617.785} C_VEL
LIN {X 0,Y 389.278,Z 758.694,A -85,B 0,C 180,E1 -11619.349,E2 -11619.349} C_VEL
LIN {X 0,Y 389.652,Z 750.707,A -85,B 0,C 180,E1 -11620.915,E2 -11620.915} C_VEL
LIN {X 0,Y 390.146,Z 742.49,A -85,B 0,C 180,E1 -11622.218,E2 -11622.218} C_VEL
LIN {X 0,Y 390.917,Z 732.467,A -85,B 0,C 180,E1 -11623.514,E2 -11623.514} C_VEL
LIN {X 0,Y 391.431,Z 722.55,A -85,B 0,C 180,E1 -11624.556,E2 -11624.556} C_VEL
LIN {X 0,Y 392.207,Z 710.017,A -85,B 0,C 180,E1 -11625.59,E2 -11625.59} C_VEL
LIN {X 0,Y 392.917,Z 697.76,A -85,B 0,C 180,E1 -11626.361,E2 -11626.361} C_VEL
LIN {X 0,Y 394.001,Z 681.29,A -85,B 0,C 180,E1 -11627.248,E2 -11627.248} C_VEL
LIN {X 0,Y 394.561,Z 668.613,A -85,B 0,C 180,E1 -11627.725,E2 -11627.725} C_VEL
LIN {X 0,Y 394.875,Z 652.464,A -85,B 0,C 180,E1 -11628.079,E2 -11628.079} C_VEL
LIN {X 0,Y 395.462,Z 594.18,A -85,B 0,C 180,E1 -11629.138,E2 -11629.138} C_VEL
LIN {X 0,Y 391.45,Z 554.419,A -85,B 0,C 180,E1 -11630.08,E2 -11630.08} C_VEL
LIN {X 0,Y 391.432,Z 552.883,A -85,B 0,C 180,E1 -11630.218,E2 -11630.218} C_VEL
LIN {X 0,Y 392.867,Z 529.579,A -85,B 0,C 180,E1 -11633.915,E2 -11633.915} C_VEL
LIN {X 0,Y 394.431,Z 507.778,A -85,B 0,C 180,E1 -11637.401,E2 -11637.401} C_VEL
LIN {X 0,Y 395.064,Z 499.719,A -85,B 0,C 180,E1 -11638.704,E2 -11638.704} C_VEL
LIN {X 0,Y 393.107,Z 489.595,A -85,B 0,C 180,E1 -11640.489,E2 -11640.489} C_VEL
LIN {X 0,Y 390.108,Z 476.014,A -85,B 0,C 180,E1 -11643.02,E2 -11643.02} C_VEL
LIN {X 0,Y 390.047,Z 475.898,A -85,B 0,C 180,E1 -11646.482,E2 -11646.482} C_VEL
LIN {X 0,Y 390.028,Z 475.897,A -85,B 0,C 180,E1 -11649.21,E2 -11649.21} C_VEL
LIN {X 0,Y 390.024,Z 475.903,A -85,B 0,C 180,E1 -11652.371,E2 -11652.371} C_VEL
LIN {X 0,Y 390.035,Z 475.896,A -85,B 0,C 180,E1 -11655.352,E2 -11655.352} C_VEL
LIN {X 0,Y 390.013,Z 475.906,A -85,B 0,C 180,E1 -11658.184,E2 -11658.184} C_VEL
LIN {X 0,Y 390.049,Z 475.896,A -85,B 0,C 180,E1 -11660.902,E2 -11660.902} C_VEL
LIN {X 0,Y 390.074,Z 475.893,A -85,B 0,C 180,E1 -11664.792,E2 -11664.792} C_VEL
LIN {X 0,Y 390.013,Z 475.904,A -85,B 0,C 180,E1 -11668.494,E2 -11668.494} C_VEL
LIN {X 0,Y 390.106,Z 475.891,A -85,B 0,C 180,E1 -11672.069,E2 -11672.069} C_VEL
LIN {X 0,Y 390.064,Z 475.893,A -85,B 0,C 180,E1 -11675.518,E2 -11675.518} C_VEL
LIN {X 0,Y 390.05,Z 475.896,A -85,B 0,C 180,E1 -11678.877,E2 -11678.877} C_VEL
LIN {X 0,Y 390.115,Z 475.891,A -85,B 0,C 180,E1 -11682.166,E2 -11682.166} C_VEL
LIN {X 0,Y 390.13,Z 475.884,A -85,B 0,C 180,E1 -11685.392,E2 -11685.392} C_VEL
LIN {X 0,Y 390.136,Z 475.89,A -85,B 0,C 180,E1 -11688.57,E2 -11688.57} C_VEL
LIN {X 0,Y 390.33,Z 475.861,A -85,B 0,C 180,E1 -11691.993,E2 -11691.993} C_VEL
LIN {X 0,Y 390.21,Z 475.878,A -85,B 0,C 180,E1 -11694.833,E2 -11694.833} C_VEL
LIN {X 0,Y 390.404,Z 475.852,A -85,B 0,C 180,E1 -11697.936,E2 -11697.936} C_VEL
LIN {X 0,Y 390.535,Z 475.836,A -85,B 0,C 180,E1 -11700,E2 -11700} C_VEL
LIN {X 0,Y 390.3,Z 475.865,A -85,B 0,C 180,E1 -11703.096,E2 -11703.096} C_VEL
LIN {X 0,Y 390.292,Z 475.864,A -85,B 0,C 180,E1 -11706.705,E2 -11706.705} C_VEL
LIN {X 0,Y 390.191,Z 475.878,A -85,B 0,C 180,E1 -11709.329,E2 -11709.329} C_VEL
LIN {X 0,Y 390.157,Z 475.886,A -85,B 0,C 180,E1 -11712.483,E2 -11712.483} C_VEL
LIN {X 0,Y 390.125,Z 475.885,A -85,B 0,C 180,E1 -11715.677,E2 -11715.677} C_VEL
LIN {X 0,Y 390.091,Z 475.894,A -85,B 0,C 180,E1 -11718.922,E2 -11718.922} C_VEL
LIN {X 0,Y 390.026,Z 475.899,A -85,B 0,C 180,E1 -11722.235,E2 -11722.235} C_VEL
LIN {X 0,Y 390.105,Z 475.888,A -85,B 0,C 180,E1 -11725.744,E2 -11725.744} C_VEL
LIN {X 0,Y 390.045,Z 475.898,A -85,B 0,C 180,E1 -11729.11,E2 -11729.11} C_VEL
LIN {X 0,Y 390.029,Z 475.904,A -85,B 0,C 180,E1 -11732.722,E2 -11732.722} C_VEL
LIN {X 0,Y 390.044,Z 475.895,A -85,B 0,C 180,E1 -11735.827,E2 -11735.827} C_VEL
LIN {X 0,Y 390.058,Z 475.896,A -85,B 0,C 180,E1 -11739.219,E2 -11739.219} C_VEL
LIN {X 0,Y 390.033,Z 475.899,A -85,B 0,C 180,E1 -11742.376,E2 -11742.376} C_VEL
LIN {X 0,Y 390.091,Z 475.89,A -85,B 0,C 180,E1 -11746.108,E2 -11746.108} C_VEL
LIN {X 0,Y 390.073,Z 475.896,A -85,B 0,C 180,E1 -11749.175,E2 -11749.175} C_VEL
LIN {X 0,Y 390.05,Z 475.896,A -85,B 0,C 180,E1 -11752.447,E2 -11752.447} C_VEL
LIN {X 0,Y 390.058,Z 475.893,A -85,B 0,C 180,E1 -11756.047,E2 -11756.047} C_VEL
LIN {X 0,Y 390.038,Z 475.896,A -85,B 0,C 180,E1 -11759.87,E2 -11759.87} C_VEL
LIN {X 0,Y 390.106,Z 475.892,A -85,B 0,C 180,E1 -11763.233,E2 -11763.233} C_VEL
LIN {X 0,Y 390.1,Z 475.892,A -85,B 0,C 180,E1 -11766.752,E2 -11766.752} C_VEL
LIN {X 0,Y 390.098,Z 475.889,A -85,B 0,C 180,E1 -11769.985,E2 -11769.985} C_VEL
LIN {X 0,Y 390.133,Z 475.889,A -85,B 0,C 180,E1 -11773.25,E2 -11773.25} C_VEL
LIN {X 0,Y 390.19,Z 475.879,A -85,B 0,C 180,E1 -11776.563,E2 -11776.563} C_VEL
LIN {X 0,Y 390.202,Z 475.882,A -85,B 0,C 180,E1 -11780.673,E2 -11780.673} C_VEL
LIN {X 0,Y 390.316,Z 475.866,A -85,B 0,C 180,E1 -11782.761,E2 -11782.761} C_VEL
LIN {X 0,Y 390.312,Z 476.078,A -85,B 0,C 180,E1 -11784.513,E2 -11784.513} C_VEL
LIN {X 0,Y 390.528,Z 477.186,A -85,B 0,C 180,E1 -11784.677,E2 -11784.677} C_VEL
LIN {X 0,Y 396.139,Z 492.75,A -85,B 0,C 180,E1 -11785.234,E2 -11785.234} C_VEL
LIN {X 0,Y 395.514,Z 555.678,A -85,B 0,C 180,E1 -11786.393,E2 -11786.393} C_VEL
LIN {X 0,Y 395.47,Z 568.737,A -85,B 0,C 180,E1 -11786.802,E2 -11786.802} C_VEL
LIN {X 0,Y 395.17,Z 582.115,A -85,B 0,C 180,E1 -11787.453,E2 -11787.453} C_VEL
LIN {X 0,Y 394.77,Z 593.608,A -85,B 0,C 180,E1 -11788.216,E2 -11788.216} C_VEL
LIN {X 0,Y 394.252,Z 604.64,A -85,B 0,C 180,E1 -11789.157,E2 -11789.157} C_VEL
LIN {X 0,Y 393.57,Z 615.137,A -85,B 0,C 180,E1 -11790.286,E2 -11790.286} C_VEL
LIN {X 0,Y 392.969,Z 624.552,A -85,B 0,C 180,E1 -11791.539,E2 -11791.539} C_VEL
LIN {X 0,Y 392.331,Z 632.5,A -85,B 0,C 180,E1 -11792.825,E2 -11792.825} C_VEL
LIN {X 0,Y 391.717,Z 640.298,A -85,B 0,C 180,E1 -11794.375,E2 -11794.375} C_VEL
LIN {X 0,Y 391.284,Z 645.588,A -85,B 0,C 180,E1 -11795.671,E2 -11795.671} C_VEL
LIN {X 0,Y 390.918,Z 650.756,A -85,B 0,C 180,E1 -11797.231,E2 -11797.231} C_VEL
LIN {X 0,Y 390.587,Z 654.788,A -85,B 0,C 180,E1 -11798.799,E2 -11798.799} C_VEL
LIN {X 0,Y 390.303,Z 657.792,A -85,B 0,C 180,E1 -11800.375,E2 -11800.375} C_VEL
LIN {X 0,Y 390.147,Z 659.892,A -85,B 0,C 180,E1 -11802.105,E2 -11802.105} C_VEL
LIN {X 0,Y 389.482,Z 660.706,A -85,B 0,C 180,E1 -11802.96,E2 -11802.96} C_VEL
LIN {X 0,Y 386.65,Z 661.598,A -85,B 0,C 180,E1 -11804.357,E2 -11804.357} C_VEL
LIN {X 0,Y 383.89,Z 661.841,A -85,B 0,C 180,E1 -11805.777,E2 -11805.777} C_VEL
LIN {X 0,Y 383.352,Z 661.424,A -85,B 0,C 180,E1 -11806.656,E2 -11806.656} C_VEL
LIN {X 0,Y 383.621,Z 660.072,A -85,B 0,C 180,E1 -11808.148,E2 -11808.148} C_VEL
LIN {X 0,Y 383.851,Z 658.519,A -85,B 0,C 180,E1 -11809.244,E2 -11809.244} C_VEL
LIN {X 0,Y 384.483,Z 654.592,A -85,B 0,C 180,E1 -11811.215,E2 -11811.215} C_VEL
LIN {X 0,Y 385.235,Z 649.254,A -85,B 0,C 180,E1 -11813.095,E2 -11813.095} C_VEL
LIN {X 0,Y 386.078,Z 643.115,A -85,B 0,C 180,E1 -11814.753,E2 -11814.753} C_VEL
LIN {X 0,Y 387.074,Z 635.343,A -85,B 0,C 180,E1 -11816.415,E2 -11816.415} C_VEL
LIN {X 0,Y 388.031,Z 626.932,A -85,B 0,C 180,E1 -11817.847,E2 -11817.847} C_VEL
LIN {X 0,Y 388.955,Z 617.131,A -85,B 0,C 180,E1 -11819.202,E2 -11819.202} C_VEL
LIN {X 0,Y 389.895,Z 607.103,A -85,B 0,C 180,E1 -11820.314,E2 -11820.314} C_VEL
LIN {X 0,Y 390.676,Z 595.992,A -85,B 0,C 180,E1 -11821.297,E2 -11821.297} C_VEL
LIN {X 0,Y 391.243,Z 584.042,A -85,B 0,C 180,E1 -11822.117,E2 -11822.117} C_VEL
LIN {X 0,Y 391.641,Z 571.517,A -85,B 0,C 180,E1 -11822.75,E2 -11822.75} C_VEL
LIN {X 0,Y 391.76,Z 559.231,A -85,B 0,C 180,E1 -11823.165,E2 -11823.165} C_VEL
LIN {X 0,Y 392.135,Z 520.655,A -85,B 0,C 180,E1 -11823.922,E2 -11823.922} C_VEL
LIN {X 0,Y 392.415,Z 497.795,A -85,B 0,C 180,E1 -11824.359,E2 -11824.359} C_VEL
LIN {X 0,Y 384.185,Z 479.836,A -85,B 0,C 180,E1 -11825.297,E2 -11825.297} C_VEL
LIN {X 0,Y 383.199,Z 477.567,A -85,B 0,C 180,E1 -11825.455,E2 -11825.455} C_VEL
LIN {X 0,Y 383.051,Z 476.82,A -85,B 0,C 180,E1 -11825.695,E2 -11825.695} C_VEL
LIN {X 0,Y 383.017,Z 476.768,A -85,B 0,C 180,E1 -11829.588,E2 -11829.588} C_VEL
LIN {X 0,Y 383.01,Z 476.768,A -85,B 0,C 180,E1 -11832.78,E2 -11832.78} C_VEL
LIN {X 0,Y 383.002,Z 476.777,A -85,B 0,C 180,E1 -11835.79,E2 -11835.79} C_VEL
LIN {X 0,Y 383.027,Z 476.976,A -85,B 0,C 180,E1 -11838.457,E2 -11838.457} C_VEL
LIN {X 0,Y 386.089,Z 490.553,A -85,B 0,C 180,E1 -11841.108,E2 -11841.108} C_VEL
LIN {X 0,Y 387.334,Z 498.095,A -85,B 0,C 180,E1 -11842.533,E2 -11842.533} C_VEL
LIN {X 0,Y 386.415,Z 517.986,A -85,B 0,C 180,E1 -11846.026,E2 -11846.026} C_VEL
LIN {X 0,Y 386.244,Z 522.524,A -85,B 0,C 180,E1 -11846.796,E2 -11846.796} C_VEL
LIN {X 0,Y 389.435,Z 543.42,A -85,B 0,C 180,E1 -11847.444,E2 -11847.444} C_VEL
LIN {X 0,Y 387.56,Z 633.125,A -85,B 0,C 180,E1 -11849.411,E2 -11849.411} C_VEL
LIN {X 0,Y 387.14,Z 646.254,A -85,B 0,C 180,E1 -11849.902,E2 -11849.902} C_VEL
LIN {X 0,Y 386.568,Z 659.113,A -85,B 0,C 180,E1 -11850.602,E2 -11850.602} C_VEL
LIN {X 0,Y 385.95,Z 671.138,A -85,B 0,C 180,E1 -11851.472,E2 -11851.472} C_VEL
LIN {X 0,Y 385.152,Z 682.847,A -85,B 0,C 180,E1 -11852.565,E2 -11852.565} C_VEL
LIN {X 0,Y 384.443,Z 692.701,A -85,B 0,C 180,E1 -11853.706,E2 -11853.706} C_VEL
LIN {X 0,Y 383.764,Z 702.396,A -85,B 0,C 180,E1 -11855.09,E2 -11855.09} C_VEL
LIN {X 0,Y 383.154,Z 711.052,A -85,B 0,C 180,E1 -11856.619,E2 -11856.619} C_VEL
LIN {X 0,Y 382.632,Z 718.127,A -85,B 0,C 180,E1 -11858.165,E2 -11858.165} C_VEL
LIN {X 0,Y 382.283,Z 723.6,A -85,B 0,C 180,E1 -11859.656,E2 -11859.656} C_VEL
LIN {X 0,Y 381.995,Z 728.135,A -85,B 0,C 180,E1 -11861.218,E2 -11861.218} C_VEL
LIN {X 0,Y 381.783,Z 732.294,A -85,B 0,C 180,E1 -11863.188,E2 -11863.188} C_VEL
LIN {X 0,Y 381.587,Z 734.828,A -85,B 0,C 180,E1 -11865.058,E2 -11865.058} C_VEL
LIN {X 0,Y 381.579,Z 735.643,A -85,B 0,C 180,E1 -11866.147,E2 -11866.147} C_VEL
LIN {X 0,Y 381.691,Z 736.069,A -85,B 0,C 180,E1 -11867.396,E2 -11867.396} C_VEL
LIN {X 0,Y 381.701,Z 735.996,A -85,B 0,C 180,E1 -11868.315,E2 -11868.315} C_VEL
LIN {X 0,Y 381.725,Z 735.481,A -85,B 0,C 180,E1 -11869.391,E2 -11869.391} C_VEL
LIN {X 0,Y 381.829,Z 734.551,A -85,B 0,C 180,E1 -11870.465,E2 -11870.465} C_VEL
LIN {X 0,Y 382.005,Z 733.191,A -85,B 0,C 180,E1 -11871.537,E2 -11871.537} C_VEL
LIN {X 0,Y 382.298,Z 730.382,A -85,B 0,C 180,E1 -11873.089,E2 -11873.089} C_VEL
LIN {X 0,Y 382.627,Z 726.284,A -85,B 0,C 180,E1 -11874.731,E2 -11874.731} C_VEL
LIN {X 0,Y 383.138,Z 721.101,A -85,B 0,C 180,E1 -11876.319,E2 -11876.319} C_VEL
LIN {X 0,Y 383.781,Z 714.599,A -85,B 0,C 180,E1 -11877.901,E2 -11877.901} C_VEL
LIN {X 0,Y 384.672,Z 706.5,A -85,B 0,C 180,E1 -11879.477,E2 -11879.477} C_VEL
LIN {X 0,Y 385.499,Z 698.181,A -85,B 0,C 180,E1 -11880.784,E2 -11880.784} C_VEL
LIN {X 0,Y 386.488,Z 687.993,A -85,B 0,C 180,E1 -11882.085,E2 -11882.085} C_VEL
LIN {X 0,Y 387.448,Z 676.831,A -85,B 0,C 180,E1 -11883.226,E2 -11883.226} C_VEL
LIN {X 0,Y 388.243,Z 665.34,A -85,B 0,C 180,E1 -11884.153,E2 -11884.153} C_VEL
LIN {X 0,Y 389.063,Z 652.899,A -85,B 0,C 180,E1 -11884.923,E2 -11884.923} C_VEL
LIN {X 0,Y 389.598,Z 639.951,A -85,B 0,C 180,E1 -11885.5,E2 -11885.5} C_VEL
LIN {X 0,Y 390.037,Z 625.213,A -85,B 0,C 180,E1 -11885.915,E2 -11885.915} C_VEL
LIN {X 0,Y 392.504,Z 543.521,A -85,B 0,C 180,E1 -11887.845,E2 -11887.845} C_VEL
LIN {X 0,Y 389.372,Z 528.605,A -85,B 0,C 180,E1 -11888.501,E2 -11888.501} C_VEL
LIN {X 0,Y 388.701,Z 525.589,A -85,B 0,C 180,E1 -11888.677,E2 -11888.677} C_VEL
LIN {X 0,Y 389.942,Z 503.782,A -85,B 0,C 180,E1 -11892.491,E2 -11892.491} C_VEL
LIN {X 0,Y 388.764,Z 496.865,A -85,B 0,C 180,E1 -11893.859,E2 -11893.859} C_VEL
LIN {X 0,Y 386.046,Z 486.062,A -85,B 0,C 180,E1 -11896.119,E2 -11896.119} C_VEL
LIN {X 0,Y 383.085,Z 476.909,A -85,B 0,C 180,E1 -11898.207,E2 -11898.207} C_VEL
LIN {X 0,Y 383.001,Z 476.78,A -85,B 0,C 180,E1 -11901.531,E2 -11901.531} C_VEL
LIN {X 0,Y 383.058,Z 476.77,A -85,B 0,C 180,E1 -11904.96,E2 -11904.96} C_VEL
LIN {X 0,Y 383.039,Z 476.771,A -85,B 0,C 180,E1 -11908.27,E2 -11908.27} C_VEL
LIN {X 0,Y 383.018,Z 476.772,A -85,B 0,C 180,E1 -11912.149,E2 -11912.149} C_VEL
LIN {X 0,Y 383.027,Z 476.774,A -85,B 0,C 180,E1 -11914.667,E2 -11914.667} C_VEL
LIN {X 0,Y 383.007,Z 476.774,A -85,B 0,C 180,E1 -11917.903,E2 -11917.903} C_VEL
LIN {X 0,Y 382.992,Z 476.778,A -85,B 0,C 180,E1 -11921.347,E2 -11921.347} C_VEL
LIN {X 0,Y 383.004,Z 476.775,A -85,B 0,C 180,E1 -11924.303,E2 -11924.303} C_VEL
LIN {X 0,Y 383.019,Z 476.775,A -85,B 0,C 180,E1 -11927.239,E2 -11927.239} C_VEL
LIN {X 0,Y 383.021,Z 476.763,A -85,B 0,C 180,E1 -11930.413,E2 -11930.413} C_VEL
LIN {X 0,Y 383.022,Z 476.776,A -85,B 0,C 180,E1 -11934.042,E2 -11934.042} C_VEL
LIN {X 0,Y 383.069,Z 476.979,A -85,B 0,C 180,E1 -11934.995,E2 -11934.995} C_VEL
LIN {X 0,Y 386.555,Z 490.468,A -85,B 0,C 180,E1 -11937.887,E2 -11937.887} C_VEL
LIN {X 0,Y 389.077,Z 501.599,A -85,B 0,C 180,E1 -11940.117,E2 -11940.117} C_VEL
LIN {X 0,Y 389.461,Z 504.156,A -85,B 0,C 180,E1 -11940.601,E2 -11940.601} C_VEL
LIN {X 0,Y 387.436,Z 525.279,A -85,B 0,C 180,E1 -11944.19,E2 -11944.19} C_VEL
LIN {X 0,Y 385.622,Z 547.266,A -85,B 0,C 180,E1 -11947.84,E2 -11947.84} C_VEL
LIN {X 0,Y 386.368,Z 553.953,A -85,B 0,C 180,E1 -11948.259,E2 -11948.259} C_VEL
LIN {X 0,Y 388.725,Z 571.611,A -85,B 0,C 180,E1 -11948.939,E2 -11948.939} C_VEL
LIN {X 0,Y 390.724,Z 597.246,A -85,B 0,C 180,E1 -11949.774,E2 -11949.774} C_VEL
LIN {X 0,Y 389.655,Z 662.674,A -85,B 0,C 180,E1 -11951.024,E2 -11951.024} C_VEL
LIN {X 0,Y 388.895,Z 676.41,A -85,B 0,C 180,E1 -11951.494,E2 -11951.494} C_VEL
LIN {X 0,Y 387.957,Z 688.887,A -85,B 0,C 180,E1 -11952.13,E2 -11952.13} C_VEL
LIN {X 0,Y 386.955,Z 703.381,A -85,B 0,C 180,E1 -11952.969,E2 -11952.969} C_VEL
LIN {X 0,Y 385.997,Z 715.408,A -85,B 0,C 180,E1 -11953.878,E2 -11953.878} C_VEL
LIN {X 0,Y 385.057,Z 726.231,A -85,B 0,C 180,E1 -11954.923,E2 -11954.923} C_VEL
LIN {X 0,Y 384.138,Z 737.141,A -85,B 0,C 180,E1 -11956.239,E2 -11956.239} C_VEL
LIN {X 0,Y 383.381,Z 746.032,A -85,B 0,C 180,E1 -11957.56,E2 -11957.56} C_VEL
LIN {X 0,Y 382.652,Z 754.674,A -85,B 0,C 180,E1 -11959.147,E2 -11959.147} C_VEL
LIN {X 0,Y 382.207,Z 761.669,A -85,B 0,C 180,E1 -11960.739,E2 -11960.739} C_VEL
LIN {X 0,Y 381.961,Z 766.384,A -85,B 0,C 180,E1 -11962.066,E2 -11962.066} C_VEL
LIN {X 0,Y 381.777,Z 771.159,A -85,B 0,C 180,E1 -11963.759,E2 -11963.759} C_VEL
LIN {X 0,Y 381.785,Z 773.3,A -85,B 0,C 180,E1 -11964.717,E2 -11964.717} C_VEL
LIN {X 0,Y 381.759,Z 775.172,A -85,B 0,C 180,E1 -11965.775,E2 -11965.775} C_VEL
LIN {X 0,Y 381.77,Z 776.608,A -85,B 0,C 180,E1 -11966.832,E2 -11966.832} C_VEL
LIN {X 0,Y 381.867,Z 777.628,A -85,B 0,C 180,E1 -11967.889,E2 -11967.889} C_VEL
LIN {X 0,Y 381.838,Z 778.165,A -85,B 0,C 180,E1 -11968.944,E2 -11968.944} C_VEL
LIN {X 0,Y 381.914,Z 778.273,A -85,B 0,C 180,E1 -11969.998,E2 -11969.998} C_VEL
LIN {X 0,Y 381.856,Z 777.953,A -85,B 0,C 180,E1 -11971.053,E2 -11971.053} C_VEL
LIN {X 0,Y 381.87,Z 777.188,A -85,B 0,C 180,E1 -11972.108,E2 -11972.108} C_VEL
LIN {X 0,Y 381.819,Z 775.943,A -85,B 0,C 180,E1 -11973.164,E2 -11973.164} C_VEL
LIN {X 0,Y 381.835,Z 773.238,A -85,B 0,C 180,E1 -11974.749,E2 -11974.749} C_VEL
LIN {X 0,Y 381.81,Z 769.414,A -85,B 0,C 180,E1 -11976.339,E2 -11976.339} C_VEL
LIN {X 0,Y 381.957,Z 764.379,A -85,B 0,C 180,E1 -11977.93,E2 -11977.93} C_VEL
LIN {X 0,Y 382.209,Z 757.977,A -85,B 0,C 180,E1 -11979.524,E2 -11979.524} C_VEL
LIN {X 0,Y 382.637,Z 749.879,A -85,B 0,C 180,E1 -11981.118,E2 -11981.118} C_VEL
LIN {X 0,Y 383.106,Z 741.562,A -85,B 0,C 180,E1 -11982.446,E2 -11982.446} C_VEL
LIN {X 0,Y 383.863,Z 732.52,A -85,B 0,C 180,E1 -11983.632,E2 -11983.632} C_VEL
LIN {X 0,Y 384.421,Z 722.623,A -85,B 0,C 180,E1 -11984.702,E2 -11984.702} C_VEL
LIN {X 0,Y 385.205,Z 710.341,A -85,B 0,C 180,E1 -11985.745,E2 -11985.745} C_VEL
LIN {X 0,Y 385.932,Z 698.31,A -85,B 0,C 180,E1 -11986.529,E2 -11986.529} C_VEL
LIN {X 0,Y 387.185,Z 679.168,A -85,B 0,C 180,E1 -11987.562,E2 -11987.562} C_VEL
LIN {X 0,Y 387.78,Z 665.79,A -85,B 0,C 180,E1 -11988.045,E2 -11988.045} C_VEL
LIN {X 0,Y 388.142,Z 643.199,A -85,B 0,C 180,E1 -11988.506,E2 -11988.506} C_VEL
LIN {X 0,Y 388.645,Z 594.849,A -85,B 0,C 180,E1 -11989.401,E2 -11989.401} C_VEL
LIN {X 0,Y 384.606,Z 554.725,A -85,B 0,C 180,E1 -11990.365,E2 -11990.365} C_VEL
LIN {X 0,Y 384.453,Z 551.988,A -85,B 0,C 180,E1 -11990.528,E2 -11990.528} C_VEL
LIN {X 0,Y 386.083,Z 527.614,A -85,B 0,C 180,E1 -11994.471,E2 -11994.471} C_VEL
LIN {X 0,Y 387.722,Z 505.31,A -85,B 0,C 180,E1 -11998.116,E2 -11998.116} C_VEL
LIN {X 0,Y 388.047,Z 500.101,A -85,B 0,C 180,E1 -11998.976,E2 -11998.976} C_VEL
LIN {X 0,Y 384.884,Z 485.065,A -85,B 0,C 180,E1 -12001.72,E2 -12001.72} C_VEL
LIN {X 0,Y 383.064,Z 476.892,A -85,B 0,C 180,E1 -12003.308,E2 -12003.308} C_VEL
LIN {X 0,Y 383.023,Z 476.777,A -85,B 0,C 180,E1 -12006.162,E2 -12006.162} C_VEL
LIN {X 0,Y 382.967,Z 476.781,A -85,B 0,C 180,E1 -12009.961,E2 -12009.961} C_VEL
LIN {X 0,Y 382.998,Z 476.774,A -85,B 0,C 180,E1 -12012.777,E2 -12012.777} C_VEL
LIN {X 0,Y 382.988,Z 476.777,A -85,B 0,C 180,E1 -12015.787,E2 -12015.787} C_VEL
LIN {X 0,Y 382.959,Z 476.779,A -85,B 0,C 180,E1 -12018.798,E2 -12018.798} C_VEL
LIN {X 0,Y 382.983,Z 476.78,A -85,B 0,C 180,E1 -12022.096,E2 -12022.096} C_VEL
LIN {X 0,Y 383.007,Z 476.772,A -85,B 0,C 180,E1 -12025.331,E2 -12025.331} C_VEL
LIN {X 0,Y 382.972,Z 476.777,A -85,B 0,C 180,E1 -12029.08,E2 -12029.08} C_VEL
LIN {X 0,Y 383.044,Z 476.77,A -85,B 0,C 180,E1 -12032.697,E2 -12032.697} C_VEL
LIN {X 0,Y 383.038,Z 476.769,A -85,B 0,C 180,E1 -12035.038,E2 -12035.038} C_VEL
LIN {X 0,Y 382.986,Z 476.781,A -85,B 0,C 180,E1 -12038.468,E2 -12038.468} C_VEL
LIN {X 0,Y 383.05,Z 476.768,A -85,B 0,C 180,E1 -12041.825,E2 -12041.825} C_VEL
LIN {X 0,Y 383.096,Z 476.761,A -85,B 0,C 180,E1 -12045.117,E2 -12045.117} C_VEL
LIN {X 0,Y 383.086,Z 476.768,A -85,B 0,C 180,E1 -12048.357,E2 -12048.357} C_VEL
LIN {X 0,Y 383.29,Z 476.738,A -85,B 0,C 180,E1 -12051.933,E2 -12051.933} C_VEL
LIN {X 0,Y 383.182,Z 476.754,A -85,B 0,C 180,E1 -12054.738,E2 -12054.738} C_VEL
LIN {X 0,Y 383.372,Z 476.727,A -85,B 0,C 180,E1 -12057.898,E2 -12057.898} C_VEL
LIN {X 0,Y 383.505,Z 476.711,A -85,B 0,C 180,E1 -12060,E2 -12060} C_VEL
LIN {X 0,Y 383.236,Z 476.745,A -85,B 0,C 180,E1 -12063.153,E2 -12063.153} C_VEL
LIN {X 0,Y 383.251,Z 476.742,A -85,B 0,C 180,E1 -12066.701,E2 -12066.701} C_VEL
LIN {X 0,Y 383.246,Z 476.747,A -85,B 0,C 180,E1 -12068.436,E2 -12068.436} C_VEL
LIN {X 0,Y 383.084,Z 476.762,A -85,B 0,C 180,E1 -12071.642,E2 -12071.642} C_VEL
LIN {X 0,Y 383.096,Z 476.765,A -85,B 0,C 180,E1 -12074.882,E2 -12074.882} C_VEL
LIN {X 0,Y 383.075,Z 476.765,A -85,B 0,C 180,E1 -12078.173,E2 -12078.173} C_VEL
LIN {X 0,Y 382.979,Z 476.776,A -85,B 0,C 180,E1 -12081.531,E2 -12081.531} C_VEL
LIN {X 0,Y 383.039,Z 476.772,A -85,B 0,C 180,E1 -12084.961,E2 -12084.961} C_VEL
LIN {X 0,Y 383.027,Z 476.773,A -85,B 0,C 180,E1 -12088.493,E2 -12088.493} C_VEL
LIN {X 0,Y 382.996,Z 476.774,A -85,B 0,C 180,E1 -12092.151,E2 -12092.151} C_VEL
LIN {X 0,Y 383.005,Z 476.778,A -85,B 0,C 180,E1 -12094.669,E2 -12094.669} C_VEL
LIN {X 0,Y 382.988,Z 476.774,A -85,B 0,C 180,E1 -12097.905,E2 -12097.905} C_VEL
LIN {X 0,Y 382.972,Z 476.778,A -85,B 0,C 180,E1 -12101.348,E2 -12101.348} C_VEL
LIN {X 0,Y 382.999,Z 476.774,A -85,B 0,C 180,E1 -12104.307,E2 -12104.307} C_VEL
LIN {X 0,Y 383.064,Z 476.768,A -85,B 0,C 180,E1 -12107.25,E2 -12107.25} C_VEL
LIN {X 0,Y 383.013,Z 476.773,A -85,B 0,C 180,E1 -12110.413,E2 -12110.413} C_VEL
LIN {X 0,Y 383.017,Z 476.771,A -85,B 0,C 180,E1 -12114.046,E2 -12114.046} C_VEL
LIN {X 0,Y 382.978,Z 476.777,A -85,B 0,C 180,E1 -12117.579,E2 -12117.579} C_VEL
LIN {X 0,Y 382.984,Z 476.775,A -85,B 0,C 180,E1 -12120.302,E2 -12120.302} C_VEL
LIN {X 0,Y 383.073,Z 476.764,A -85,B 0,C 180,E1 -12124.022,E2 -12124.022} C_VEL
LIN {X 0,Y 383.002,Z 476.776,A -85,B 0,C 180,E1 -12127.337,E2 -12127.337} C_VEL
LIN {X 0,Y 383.055,Z 476.769,A -85,B 0,C 180,E1 -12130.718,E2 -12130.718} C_VEL
LIN {X 0,Y 383.075,Z 476.763,A -85,B 0,C 180,E1 -12134.028,E2 -12134.028} C_VEL
LIN {X 0,Y 383.132,Z 476.761,A -85,B 0,C 180,E1 -12137.286,E2 -12137.286} C_VEL
LIN {X 0,Y 383.148,Z 476.76,A -85,B 0,C 180,E1 -12140.5,E2 -12140.5} C_VEL
LIN {X 0,Y 383.271,Z 476.745,A -85,B 0,C 180,E1 -12142.627,E2 -12142.627} C_VEL
LIN {X 0,Y 383.303,Z 476.96,A -85,B 0,C 180,E1 -12144.214,E2 -12144.214} C_VEL
LIN {X 0,Y 383.45,Z 477.799,A -85,B 0,C 180,E1 -12144.361,E2 -12144.361} C_VEL
LIN {X 0,Y 389.374,Z 494.558,A -85,B 0,C 180,E1 -12144.969,E2 -12144.969} C_VEL
LIN {X 0,Y 388.679,Z 554.996,A -85,B 0,C 180,E1 -12146.096,E2 -12146.096} C_VEL
LIN {X 0,Y 388.663,Z 568.233,A -85,B 0,C 180,E1 -12146.494,E2 -12146.494} C_VEL
LIN {X 0,Y 388.415,Z 580.883,A -85,B 0,C 180,E1 -12147.085,E2 -12147.085} C_VEL
LIN {X 0,Y 387.936,Z 593.73,A -85,B 0,C 180,E1 -12147.925,E2 -12147.925} C_VEL
LIN {X 0,Y 387.45,Z 604.391,A -85,B 0,C 180,E1 -12148.832,E2 -12148.832} C_VEL
LIN {X 0,Y 386.715,Z 615.356,A -85,B 0,C 180,E1 -12150.002,E2 -12150.002} C_VEL
LIN {X 0,Y 386.071,Z 625.089,A -85,B 0,C 180,E1 -12151.306,E2 -12151.306} C_VEL
LIN {X 0,Y 385.41,Z 633.109,A -85,B 0,C 180,E1 -12152.615,E2 -12152.615} C_VEL
LIN {X 0,Y 384.774,Z 640.982,A -85,B 0,C 180,E1 -12154.192,E2 -12154.192} C_VEL
LIN {X 0,Y 384.239,Z 647.282,A -85,B 0,C 180,E1 -12155.775,E2 -12155.775} C_VEL
LIN {X 0,Y 383.856,Z 652.287,A -85,B 0,C 180,E1 -12157.365,E2 -12157.365} C_VEL
LIN {X 0,Y 383.519,Z 656.188,A -85,B 0,C 180,E1 -12158.963,E2 -12158.963} C_VEL
LIN {X 0,Y 383.253,Z 659.07,A -85,B 0,C 180,E1 -12160.568,E2 -12160.568} C_VEL
LIN {X 0,Y 383.121,Z 661.406,A -85,B 0,C 180,E1 -12162.718,E2 -12162.718} C_VEL
LIN {X 0,Y 383.129,Z 661.977,A -85,B 0,C 180,E1 -12163.798,E2 -12163.798} C_VEL
LIN {X 0,Y 383.151,Z 662.109,A -85,B 0,C 180,E1 -12164.882,E2 -12164.882} C_VEL
LIN {X 0,Y 383.352,Z 661.424,A -85,B 0,C 180,E1 -12166.656,E2 -12166.656} C_VEL
LIN {X 0,Y 382.846,Z 660.86,A -85,B 0,C 180,E1 -12167.532,E2 -12167.532} C_VEL
LIN {X 0,Y 380.29,Z 659.592,A -85,B 0,C 180,E1 -12168.96,E2 -12168.96} C_VEL
LIN {X 0,Y 378.196,Z 658.111,A -85,B 0,C 180,E1 -12170.098,E2 -12170.098} C_VEL
LIN {X 0,Y 377.464,Z 656.576,A -85,B 0,C 180,E1 -12170.958,E2 -12170.958} C_VEL
LIN {X 0,Y 377.498,Z 655.945,A -85,B 0,C 180,E1 -12171.243,E2 -12171.243} C_VEL
LIN {X 0,Y 378.21,Z 651.368,A -85,B 0,C 180,E1 -12172.97,E2 -12172.97} C_VEL
LIN {X 0,Y 379.183,Z 644.648,A -85,B 0,C 180,E1 -12174.877,E2 -12174.877} C_VEL
LIN {X 0,Y 380.254,Z 636.711,A -85,B 0,C 180,E1 -12176.63,E2 -12176.63} C_VEL
LIN {X 0,Y 381.232,Z 628.634,A -85,B 0,C 180,E1 -12178.051,E2 -12178.051} C_VEL
LIN {X 0,Y 382.245,Z 618.715,A -85,B 0,C 180,E1 -12179.463,E2 -12179.463} C_VEL
LIN {X 0,Y 383.184,Z 609.18,A -85,B 0,C 180,E1 -12180.555,E2 -12180.555} C_VEL
LIN {X 0,Y 384.059,Z 597.967,A -85,B 0,C 180,E1 -12181.59,E2 -12181.59} C_VEL
LIN {X 0,Y 384.668,Z 586.143,A -85,B 0,C 180,E1 -12182.434,E2 -12182.434} C_VEL
LIN {X 0,Y 385.133,Z 572.939,A -85,B 0,C 180,E1 -12183.125,E2 -12183.125} C_VEL
LIN {X 0,Y 385.291,Z 560.919,A -85,B 0,C 180,E1 -12183.548,E2 -12183.548} C_VEL
LIN {X 0,Y 385.61,Z 524.223,A -85,B 0,C 180,E1 -12184.289,E2 -12184.289} C_VEL
LIN {X 0,Y 386.017,Z 499.709,A -85,B 0,C 180,E1 -12184.759,E2 -12184.759} C_VEL
LIN {X 0,Y 376.96,Z 480.437,A -85,B 0,C 180,E1 -12185.815,E2 -12185.815} C_VEL
LIN {X 0,Y 376.098,Z 478.282,A -85,B 0,C 180,E1 -12185.988,E2 -12185.988} C_VEL
LIN {X 0,Y 376.005,Z 477.698,A -85,B 0,C 180,E1 -12186.215,E2 -12186.215} C_VEL
LIN {X 0,Y 375.992,Z 477.643,A -85,B 0,C 180,E1 -12189.972,E2 -12189.972} C_VEL
LIN {X 0,Y 375.934,Z 477.657,A -85,B 0,C 180,E1 -12193.767,E2 -12193.767} C_VEL
LIN {X 0,Y 375.956,Z 477.656,A -85,B 0,C 180,E1 -12197.704,E2 -12197.704} C_VEL
LIN {X 0,Y 376.006,Z 477.871,A -85,B 0,C 180,E1 -12198.174,E2 -12198.174} C_VEL
LIN {X 0,Y 379.322,Z 492.709,A -85,B 0,C 180,E1 -12201.095,E2 -12201.095} C_VEL
LIN {X 0,Y 380.429,Z 499.758,A -85,B 0,C 180,E1 -12202.437,E2 -12202.437} C_VEL
LIN {X 0,Y 379.484,Z 519.517,A -85,B 0,C 180,E1 -12205.929,E2 -12205.929} C_VEL
LIN {X 0,Y 379.353,Z 523.081,A -85,B 0,C 180,E1 -12206.511,E2 -12206.511} C_VEL
LIN {X 0,Y 382.607,Z 543.098,A -85,B 0,C 180,E1 -12207.141,E2 -12207.141} C_VEL
LIN {X 0,Y 380.66,Z 633.432,A -85,B 0,C 180,E1 -12209.181,E2 -12209.181} C_VEL
LIN {X 0,Y 380.209,Z 646.539,A -85,B 0,C 180,E1 -12209.678,E2 -12209.678} C_VEL
LIN {X 0,Y 379.621,Z 659.682,A -85,B 0,C 180,E1 -12210.41,E2 -12210.41} C_VEL
LIN {X 0,Y 378.946,Z 671.98,A -85,B 0,C 180,E1 -12211.323,E2 -12211.323} C_VEL
LIN {X 0,Y 378.123,Z 683.959,A -85,B 0,C 180,E1 -12212.473,E2 -12212.473} C_VEL
LIN {X 0,Y 377.333,Z 694.526,A -85,B 0,C 180,E1 -12213.746,E2 -12213.746} C_VEL
LIN {X 0,Y 376.626,Z 704.063,A -85,B 0,C 180,E1 -12215.175,E2 -12215.175} C_VEL
LIN {X 0,Y 376.082,Z 711.72,A -85,B 0,C 180,E1 -12216.574,E2 -12216.574} C_VEL
LIN {X 0,Y 375.594,Z 718.237,A -85,B 0,C 180,E1 -12218.023,E2 -12218.023} C_VEL
LIN {X 0,Y 375.231,Z 723.554,A -85,B 0,C 180,E1 -12219.474,E2 -12219.474} C_VEL
LIN {X 0,Y 374.963,Z 727.634,A -85,B 0,C 180,E1 -12220.853,E2 -12220.853} C_VEL
LIN {X 0,Y 374.772,Z 731.516,A -85,B 0,C 180,E1 -12222.54,E2 -12222.54} C_VEL
LIN {X 0,Y 374.625,Z 733.434,A -85,B 0,C 180,E1 -12223.657,E2 -12223.657} C_VEL
LIN {X 0,Y 374.507,Z 734.873,A -85,B 0,C 180,E1 -12224.769,E2 -12224.769} C_VEL
LIN {X 0,Y 374.497,Z 735.877,A -85,B 0,C 180,E1 -12225.88,E2 -12225.88} C_VEL
LIN {X 0,Y 374.591,Z 736.453,A -85,B 0,C 180,E1 -12227.326,E2 -12227.326} C_VEL
LIN {X 0,Y 374.647,Z 736.114,A -85,B 0,C 180,E1 -12229.188,E2 -12229.188} C_VEL
LIN {X 0,Y 374.746,Z 735.288,A -85,B 0,C 180,E1 -12230.283,E2 -12230.283} C_VEL
LIN {X 0,Y 374.898,Z 734.044,A -85,B 0,C 180,E1 -12231.375,E2 -12231.375} C_VEL
LIN {X 0,Y 375.229,Z 731.211,A -85,B 0,C 180,E1 -12233.076,E2 -12233.076} C_VEL
LIN {X 0,Y 375.562,Z 727.593,A -85,B 0,C 180,E1 -12234.632,E2 -12234.632} C_VEL
LIN {X 0,Y 376.076,Z 722.683,A -85,B 0,C 180,E1 -12236.25,E2 -12236.25} C_VEL
LIN {X 0,Y 376.741,Z 716.449,A -85,B 0,C 180,E1 -12237.862,E2 -12237.862} C_VEL
LIN {X 0,Y 377.645,Z 708.634,A -85,B 0,C 180,E1 -12239.467,E2 -12239.467} C_VEL
LIN {X 0,Y 378.523,Z 700.677,A -85,B 0,C 180,E1 -12240.798,E2 -12240.798} C_VEL
LIN {X 0,Y 379.525,Z 691.015,A -85,B 0,C 180,E1 -12242.123,E2 -12242.123} C_VEL
LIN {X 0,Y 380.606,Z 679.88,A -85,B 0,C 180,E1 -12243.344,E2 -12243.344} C_VEL
LIN {X 0,Y 381.506,Z 668.28,A -85,B 0,C 180,E1 -12244.358,E2 -12244.358} C_VEL
LIN {X 0,Y 382.407,Z 655.427,A -85,B 0,C 180,E1 -12245.207,E2 -12245.207} C_VEL
LIN {X 0,Y 382.997,Z 642.73,A -85,B 0,C 180,E1 -12245.826,E2 -12245.826} C_VEL
LIN {X 0,Y 383.459,Z 629.392,A -85,B 0,C 180,E1 -12246.248,E2 -12246.248} C_VEL
LIN {X 0,Y 386.25,Z 544.714,A -85,B 0,C 180,E1 -12248.305,E2 -12248.305} C_VEL
LIN {X 0,Y 382.681,Z 528.128,A -85,B 0,C 180,E1 -12249.079,E2 -12249.079} C_VEL
LIN {X 0,Y 382.244,Z 526.06,A -85,B 0,C 180,E1 -12249.225,E2 -12249.225} C_VEL
LIN {X 0,Y 383.437,Z 506.332,A -85,B 0,C 180,E1 -12252.706,E2 -12252.706} C_VEL
LIN {X 0,Y 382.641,Z 500.801,A -85,B 0,C 180,E1 -12253.814,E2 -12253.814} C_VEL
LIN {X 0,Y 380.043,Z 490.08,A -85,B 0,C 180,E1 -12256.105,E2 -12256.105} C_VEL
LIN {X 0,Y 377.168,Z 481.143,A -85,B 0,C 180,E1 -12258.133,E2 -12258.133} C_VEL
LIN {X 0,Y 376.047,Z 477.788,A -85,B 0,C 180,E1 -12258.985,E2 -12258.985} C_VEL
LIN {X 0,Y 375.965,Z 477.654,A -85,B 0,C 180,E1 -12261.955,E2 -12261.955} C_VEL
LIN {X 0,Y 376.013,Z 477.648,A -85,B 0,C 180,E1 -12265.461,E2 -12265.461} C_VEL
LIN {X 0,Y 375.97,Z 477.655,A -85,B 0,C 180,E1 -12269.08,E2 -12269.08} C_VEL
LIN {X 0,Y 375.958,Z 477.656,A -85,B 0,C 180,E1 -12272.828,E2 -12272.828} C_VEL
LIN {X 0,Y 375.966,Z 477.652,A -85,B 0,C 180,E1 -12275.415,E2 -12275.415} C_VEL
LIN {X 0,Y 375.982,Z 477.649,A -85,B 0,C 180,E1 -12278.27,E2 -12278.27} C_VEL
LIN {X 0,Y 375.943,Z 477.656,A -85,B 0,C 180,E1 -12281.6,E2 -12281.6} C_VEL
LIN {X 0,Y 375.935,Z 477.658,A -85,B 0,C 180,E1 -12285.268,E2 -12285.268} C_VEL
LIN {X 0,Y 375.942,Z 477.655,A -85,B 0,C 180,E1 -12288.398,E2 -12288.398} C_VEL
LIN {X 0,Y 375.979,Z 477.625,A -85,B 0,C 180,E1 -12291.729,E2 -12291.729} C_VEL
LIN {X 0,Y 376.017,Z 477.865,A -85,B 0,C 180,E1 -12294.507,E2 -12294.507} C_VEL
LIN {X 0,Y 379.317,Z 490.404,A -85,B 0,C 180,E1 -12297.284,E2 -12297.284} C_VEL
LIN {X 0,Y 382.139,Z 502.691,A -85,B 0,C 180,E1 -12299.813,E2 -12299.813} C_VEL
LIN {X 0,Y 382.596,Z 506.624,A -85,B 0,C 180,E1 -12300.567,E2 -12300.567} C_VEL
LIN {X 0,Y 380.415,Z 528.018,A -85,B 0,C 180,E1 -12304.267,E2 -12304.267} C_VEL
LIN {X 0,Y 378.949,Z 544.883,A -85,B 0,C 180,E1 -12307.14,E2 -12307.14} C_VEL
LIN {X 0,Y 379.625,Z 551.727,A -85,B 0,C 180,E1 -12307.594,E2 -12307.594} C_VEL
LIN {X 0,Y 381.199,Z 562.509,A -85,B 0,C 180,E1 -12308.086,E2 -12308.086} C_VEL
LIN {X 0,Y 383.149,Z 580.606,A -85,B 0,C 180,E1 -12308.755,E2 -12308.755} C_VEL
LIN {X 0,Y 384.277,Z 599.262,A -85,B 0,C 180,E1 -12309.366,E2 -12309.366} C_VEL
LIN {X 0,Y 383.796,Z 619.048,A -85,B 0,C 180,E1 -12309.785,E2 -12309.785} C_VEL
LIN {X 0,Y 383.107,Z 661.506,A -85,B 0,C 180,E1 -12310.62,E2 -12310.62} C_VEL
LIN {X 0,Y 382.366,Z 674.474,A -85,B 0,C 180,E1 -12311.061,E2 -12311.061} C_VEL
LIN {X 0,Y 380.609,Z 697.93,A -85,B 0,C 180,E1 -12312.26,E2 -12312.26} C_VEL
LIN {X 0,Y 379.777,Z 709.359,A -85,B 0,C 180,E1 -12313.053,E2 -12313.053} C_VEL
LIN {X 0,Y 378.701,Z 721.321,A -85,B 0,C 180,E1 -12314.112,E2 -12314.112} C_VEL
LIN {X 0,Y 377.681,Z 732.006,A -85,B 0,C 180,E1 -12315.301,E2 -12315.301} C_VEL
LIN {X 0,Y 376.797,Z 740.929,A -85,B 0,C 180,E1 -12316.516,E2 -12316.516} C_VEL
LIN {X 0,Y 376.191,Z 749.086,A -85,B 0,C 180,E1 -12317.866,E2 -12317.866} C_VEL
LIN {X 0,Y 375.491,Z 757.041,A -85,B 0,C 180,E1 -12319.483,E2 -12319.483} C_VEL
LIN {X 0,Y 375.114,Z 762.491,A -85,B 0,C 180,E1 -12320.835,E2 -12320.835} C_VEL
LIN {X 0,Y 374.809,Z 767.772,A -85,B 0,C 180,E1 -12322.456,E2 -12322.456} C_VEL
LIN {X 0,Y 374.693,Z 771.218,A -85,B 0,C 180,E1 -12323.779,E2 -12323.779} C_VEL
LIN {X 0,Y 374.681,Z 774.846,A -85,B 0,C 180,E1 -12325.695,E2 -12325.695} C_VEL
LIN {X 0,Y 374.671,Z 776.268,A -85,B 0,C 180,E1 -12326.772,E2 -12326.772} C_VEL
LIN {X 0,Y 374.795,Z 777.261,A -85,B 0,C 180,E1 -12327.849,E2 -12327.849} C_VEL
LIN {X 0,Y 374.764,Z 777.765,A -85,B 0,C 180,E1 -12328.924,E2 -12328.924} C_VEL
LIN {X 0,Y 374.832,Z 777.85,A -85,B 0,C 180,E1 -12329.998,E2 -12329.998} C_VEL
LIN {X 0,Y 374.781,Z 777.509,A -85,B 0,C 180,E1 -12331.073,E2 -12331.073} C_VEL
LIN {X 0,Y 374.8,Z 776.695,A -85,B 0,C 180,E1 -12332.147,E2 -12332.147} C_VEL
LIN {X 0,Y 374.723,Z 775.424,A -85,B 0,C 180,E1 -12333.224,E2 -12333.224} C_VEL
LIN {X 0,Y 374.765,Z 772.668,A -85,B 0,C 180,E1 -12334.839,E2 -12334.839} C_VEL
LIN {X 0,Y 374.724,Z 768.783,A -85,B 0,C 180,E1 -12336.459,E2 -12336.459} C_VEL
LIN {X 0,Y 374.885,Z 763.681,A -85,B 0,C 180,E1 -12338.081,E2 -12338.081} C_VEL
LIN {X 0,Y 375.156,Z 757.184,A -85,B 0,C 180,E1 -12339.705,E2 -12339.705} C_VEL
LIN {X 0,Y 375.629,Z 748.971,A -85,B 0,C 180,E1 -12341.328,E2 -12341.328} C_VEL
LIN {X 0,Y 376.115,Z 740.542,A -85,B 0,C 180,E1 -12342.681,E2 -12342.681} C_VEL
LIN {X 0,Y 376.822,Z 732.459,A -85,B 0,C 180,E1 -12343.755,E2 -12343.755} C_VEL
LIN {X 0,Y 377.485,Z 721.486,A -85,B 0,C 180,E1 -12344.955,E2 -12344.955} C_VEL
LIN {X 0,Y 378.207,Z 710.468,A -85,B 0,C 180,E1 -12345.906,E2 -12345.906} C_VEL
LIN {X 0,Y 378.95,Z 698.585,A -85,B 0,C 180,E1 -12346.704,E2 -12346.704} C_VEL
LIN {X 0,Y 380.22,Z 679.76,A -85,B 0,C 180,E1 -12347.755,E2 -12347.755} C_VEL
LIN {X 0,Y 380.817,Z 667.374,A -85,B 0,C 180,E1 -12348.248,E2 -12348.248} C_VEL
LIN {X 0,Y 381.16,Z 651.616,A -85,B 0,C 180,E1 -12348.613,E2 -12348.613} C_VEL
LIN {X 0,Y 381.786,Z 595.382,A -85,B 0,C 180,E1 -12349.671,E2 -12349.671} C_VEL
LIN {X 0,Y 377.775,Z 555.259,A -85,B 0,C 180,E1 -12350.65,E2 -12350.65} C_VEL
LIN {X 0,Y 377.508,Z 551.095,A -85,B 0,C 180,E1 -12350.857,E2 -12350.857} C_VEL
LIN {X 0,Y 379.113,Z 527.634,A -85,B 0,C 180,E1 -12354.719,E2 -12354.719} C_VEL
LIN {X 0,Y 380.838,Z 505.685,A -85,B 0,C 180,E1 -12358.369,E2 -12358.369} C_VEL
LIN {X 0,Y 381.106,Z 502.233,A -85,B 0,C 180,E1 -12358.95,E2 -12358.95} C_VEL
LIN {X 0,Y 379.78,Z 494.939,A -85,B 0,C 180,E1 -12360.281,E2 -12360.281} C_VEL
LIN {X 0,Y 376.529,Z 480.167,A -85,B 0,C 180,E1 -12363.087,E2 -12363.087} C_VEL
LIN {X 0,Y 376.016,Z 477.744,A -85,B 0,C 180,E1 -12363.619,E2 -12363.619} C_VEL
LIN {X 0,Y 375.944,Z 477.653,A -85,B 0,C 180,E1 -12366.74,E2 -12366.74} C_VEL
LIN {X 0,Y 375.93,Z 477.658,A -85,B 0,C 180,E1 -12369.959,E2 -12369.959} C_VEL
LIN {X 0,Y 375.92,Z 477.657,A -85,B 0,C 180,E1 -12373.764,E2 -12373.764} C_VEL
LIN {X 0,Y 375.925,Z 477.655,A -85,B 0,C 180,E1 -12376.809,E2 -12376.809} C_VEL
LIN {X 0,Y 375.929,Z 477.657,A -85,B 0,C 180,E1 -12380.533,E2 -12380.533} C_VEL
LIN {X 0,Y 375.952,Z 477.651,A -85,B 0,C 180,E1 -12383.494,E2 -12383.494} C_VEL
LIN {X 0,Y 375.95,Z 477.654,A -85,B 0,C 180,E1 -12385.887,E2 -12385.887} C_VEL
LIN {X 0,Y 375.953,Z 477.651,A -85,B 0,C 180,E1 -12389.686,E2 -12389.686} C_VEL
LIN {X 0,Y 376.007,Z 477.644,A -85,B 0,C 180,E1 -12393.347,E2 -12393.347} C_VEL
LIN {X 0,Y 375.981,Z 477.649,A -85,B 0,C 180,E1 -12396.887,E2 -12396.887} C_VEL
LIN {X 0,Y 375.986,Z 477.653,A -85,B 0,C 180,E1 -12400.338,E2 -12400.338} C_VEL
LIN {X 0,Y 376.015,Z 477.643,A -85,B 0,C 180,E1 -12403.718,E2 -12403.718} C_VEL
LIN {X 0,Y 376.09,Z 477.635,A -85,B 0,C 180,E1 -12407.041,E2 -12407.041} C_VEL
LIN {X 0,Y 376.106,Z 477.637,A -85,B 0,C 180,E1 -12410.318,E2 -12410.318} C_VEL
LIN {X 0,Y 376.216,Z 477.625,A -85,B 0,C 180,E1 -12412.486,E2 -12412.486} C_VEL
LIN {X 0,Y 376.155,Z 477.631,A -85,B 0,C 180,E1 -12414.639,E2 -12414.639} C_VEL
LIN {X 0,Y 376.338,Z 477.603,A -85,B 0,C 180,E1 -12417.859,E2 -12417.859} C_VEL
LIN {X 0,Y 376.474,Z 477.587,A -85,B 0,C 180,E1 -12420,E2 -12420} C_VEL
LIN {X 0,Y 376.174,Z 477.624,A -85,B 0,C 180,E1 -12423.213,E2 -12423.213} C_VEL
LIN {X 0,Y 376.214,Z 477.62,A -85,B 0,C 180,E1 -12426.693,E2 -12426.693} C_VEL
LIN {X 0,Y 376.191,Z 477.628,A -85,B 0,C 180,E1 -12428.595,E2 -12428.595} C_VEL
LIN {X 0,Y 376.036,Z 477.641,A -85,B 0,C 180,E1 -12431.863,E2 -12431.863} C_VEL
LIN {X 0,Y 376.044,Z 477.641,A -85,B 0,C 180,E1 -12435.168,E2 -12435.168} C_VEL
LIN {X 0,Y 376.01,Z 477.649,A -85,B 0,C 180,E1 -12438.526,E2 -12438.526} C_VEL
LIN {X 0,Y 375.949,Z 477.651,A -85,B 0,C 180,E1 -12441.955,E2 -12441.955} C_VEL
LIN {X 0,Y 375.992,Z 477.646,A -85,B 0,C 180,E1 -12445.462,E2 -12445.462} C_VEL
LIN {X 0,Y 375.957,Z 477.654,A -85,B 0,C 180,E1 -12449.08,E2 -12449.08} C_VEL
LIN {X 0,Y 375.936,Z 477.659,A -85,B 0,C 180,E1 -12452.829,E2 -12452.829} C_VEL
LIN {X 0,Y 375.945,Z 477.653,A -85,B 0,C 180,E1 -12455.416,E2 -12455.416} C_VEL
LIN {X 0,Y 375.963,Z 477.651,A -85,B 0,C 180,E1 -12458.272,E2 -12458.272} C_VEL
LIN {X 0,Y 375.923,Z 477.655,A -85,B 0,C 180,E1 -12461.602,E2 -12461.602} C_VEL
LIN {X 0,Y 375.969,Z 477.651,A -85,B 0,C 180,E1 -12465.262,E2 -12465.262} C_VEL
LIN {X 0,Y 375.979,Z 477.649,A -85,B 0,C 180,E1 -12468.391,E2 -12468.391} C_VEL
LIN {X 0,Y 375.963,Z 477.649,A -85,B 0,C 180,E1 -12471.914,E2 -12471.914} C_VEL
LIN {X 0,Y 375.97,Z 477.651,A -85,B 0,C 180,E1 -12475.334,E2 -12475.334} C_VEL
LIN {X 0,Y 375.949,Z 477.653,A -85,B 0,C 180,E1 -12478.44,E2 -12478.44} C_VEL
LIN {X 0,Y 375.975,Z 477.648,A -85,B 0,C 180,E1 -12482.142,E2 -12482.142} C_VEL
LIN {X 0,Y 375.999,Z 477.647,A -85,B 0,C 180,E1 -12484.541,E2 -12484.541} C_VEL
LIN {X 0,Y 375.957,Z 477.65,A -85,B 0,C 180,E1 -12488.047,E2 -12488.047} C_VEL
LIN {X 0,Y 376.003,Z 477.647,A -85,B 0,C 180,E1 -12491.475,E2 -12491.475} C_VEL
LIN {X 0,Y 376.053,Z 477.642,A -85,B 0,C 180,E1 -12494.834,E2 -12494.834} C_VEL
LIN {X 0,Y 376.046,Z 477.639,A -85,B 0,C 180,E1 -12498.138,E2 -12498.138} C_VEL
LIN {X 0,Y 376.255,Z 477.618,A -85,B 0,C 180,E1 -12501.879,E2 -12501.879} C_VEL
LIN {X 0,Y 376.295,Z 477.836,A -85,B 0,C 180,E1 -12503.901,E2 -12503.901} C_VEL
LIN {X 0,Y 376.551,Z 478.943,A -85,B 0,C 180,E1 -12504.067,E2 -12504.067} C_VEL
LIN {X 0,Y 382.543,Z 496.201,A -85,B 0,C 180,E1 -12504.692,E2 -12504.692} C_VEL
LIN {X 0,Y 381.9,Z 556.762,A -85,B 0,C 180,E1 -12505.846,E2 -12505.846} C_VEL
LIN {X 0,Y 381.806,Z 570.374,A -85,B 0,C 180,E1 -12506.275,E2 -12506.275} C_VEL
LIN {X 0,Y 381.531,Z 582.985,A -85,B 0,C 180,E1 -12506.9,E2 -12506.9} C_VEL
LIN {X 0,Y 381.065,Z 595.569,A -85,B 0,C 180,E1 -12507.756,E2 -12507.756} C_VEL
LIN {X 0,Y 380.533,Z 606.073,A -85,B 0,C 180,E1 -12508.679,E2 -12508.679} C_VEL
LIN {X 0,Y 379.852,Z 615.968,A -85,B 0,C 180,E1 -12509.757,E2 -12509.757} C_VEL
LIN {X 0,Y 379.167,Z 625.631,A -85,B 0,C 180,E1 -12511.064,E2 -12511.064} C_VEL
LIN {X 0,Y 378.371,Z 635.19,A -85,B 0,C 180,E1 -12512.663,E2 -12512.663} C_VEL
LIN {X 0,Y 377.729,Z 642.809,A -85,B 0,C 180,E1 -12514.27,E2 -12514.27} C_VEL
LIN {X 0,Y 377.194,Z 648.935,A -85,B 0,C 180,E1 -12515.884,E2 -12515.884} C_VEL
LIN {X 0,Y 376.806,Z 653.803,A -85,B 0,C 180,E1 -12517.504,E2 -12517.504} C_VEL
LIN {X 0,Y 376.453,Z 657.577,A -85,B 0,C 180,E1 -12519.132,E2 -12519.132} C_VEL
LIN {X 0,Y 376.197,Z 660.335,A -85,B 0,C 180,E1 -12520.769,E2 -12520.769} C_VEL
LIN {X 0,Y 376.088,Z 661.645,A -85,B 0,C 180,E1 -12521.864,E2 -12521.864} C_VEL
LIN {X 0,Y 376.105,Z 662.889,A -85,B 0,C 180,E1 -12523.669,E2 -12523.669} C_VEL
LIN {X 0,Y 376.169,Z 663.075,A -85,B 0,C 180,E1 -12525.165,E2 -12525.165} C_VEL
LIN {X 0,Y 376.339,Z 662.465,A -85,B 0,C 180,E1 -12526.691,E2 -12526.691} C_VEL
LIN {X 0,Y 376.677,Z 660.797,A -85,B 0,C 180,E1 -12528.494,E2 -12528.494} C_VEL
LIN {X 0,Y 377.126,Z 658.183,A -85,B 0,C 180,E1 -12530.169,E2 -12530.169} C_VEL
LIN {X 0,Y 377.498,Z 655.945,A -85,B 0,C 180,E1 -12531.243,E2 -12531.243} C_VEL
LIN {X 0,Y 377.212,Z 654.031,A -85,B 0,C 180,E1 -12532.09,E2 -12532.09} C_VEL
LIN {X 0,Y 375.032,Z 650.667,A -85,B 0,C 180,E1 -12533.471,E2 -12533.471} C_VEL
LIN {X 0,Y 372.868,Z 646.714,A -85,B 0,C 180,E1 -12534.823,E2 -12534.823} C_VEL
LIN {X 0,Y 372.607,Z 643.749,A -85,B 0,C 180,E1 -12535.614,E2 -12535.614} C_VEL
LIN {X 0,Y 373.663,Z 636.611,A -85,B 0,C 180,E1 -12537.138,E2 -12537.138} C_VEL
LIN {X 0,Y 374.769,Z 627.694,A -85,B 0,C 180,E1 -12538.677,E2 -12538.677} C_VEL
LIN {X 0,Y 375.797,Z 618.085,A -85,B 0,C 180,E1 -12540.019,E2 -12540.019} C_VEL
LIN {X 0,Y 376.778,Z 608.241,A -85,B 0,C 180,E1 -12541.121,E2 -12541.121} C_VEL
LIN {X 0,Y 377.686,Z 596.244,A -85,B 0,C 180,E1 -12542.187,E2 -12542.187} C_VEL
LIN {X 0,Y 378.343,Z 583.863,A -85,B 0,C 180,E1 -12543.029,E2 -12543.029} C_VEL
LIN {X 0,Y 378.683,Z 571.077,A -85,B 0,C 180,E1 -12543.651,E2 -12543.651} C_VEL
LIN {X 0,Y 378.807,Z 558.257,A -85,B 0,C 180,E1 -12544.053,E2 -12544.053} C_VEL
LIN {X 0,Y 379.38,Z 514.973,A -85,B 0,C 180,E1 -12544.915,E2 -12544.915} C_VEL
LIN {X 0,Y 379.521,Z 501.555,A -85,B 0,C 180,E1 -12545.183,E2 -12545.183} C_VEL
LIN {X 0,Y 371.369,Z 484.172,A -85,B 0,C 180,E1 -12546.167,E2 -12546.167} C_VEL
LIN {X 0,Y 369.071,Z 479.337,A -85,B 0,C 180,E1 -12546.492,E2 -12546.492} C_VEL
LIN {X 0,Y 368.944,Z 478.578,A -85,B 0,C 180,E1 -12546.746,E2 -12546.746} C_VEL
LIN {X 0,Y 368.914,Z 478.528,A -85,B 0,C 180,E1 -12550.372,E2 -12550.372} C_VEL
LIN {X 0,Y 368.887,Z 478.534,A -85,B 0,C 180,E1 -12553.617,E2 -12553.617} C_VEL
LIN {X 0,Y 368.92,Z 478.531,A -85,B 0,C 180,E1 -12557.391,E2 -12557.391} C_VEL
LIN {X 0,Y 368.979,Z 478.813,A -85,B 0,C 180,E1 -12557.89,E2 -12557.89} C_VEL
LIN {X 0,Y 372.422,Z 494.13,A -85,B 0,C 180,E1 -12560.932,E2 -12560.932} C_VEL
LIN {X 0,Y 373.525,Z 500.756,A -85,B 0,C 180,E1 -12562.211,E2 -12562.211} C_VEL
LIN {X 0,Y 372.511,Z 521.415,A -85,B 0,C 180,E1 -12565.899,E2 -12565.899} C_VEL
LIN {X 0,Y 372.479,Z 523.337,A -85,B 0,C 180,E1 -12566.201,E2 -12566.201} C_VEL
LIN {X 0,Y 375.769,Z 544.93,A -85,B 0,C 180,E1 -12566.888,E2 -12566.888} C_VEL
LIN {X 0,Y 373.746,Z 633.688,A -85,B 0,C 180,E1 -12568.94,E2 -12568.94} C_VEL
LIN {X 0,Y 373.304,Z 646.846,A -85,B 0,C 180,E1 -12569.449,E2 -12569.449} C_VEL
LIN {X 0,Y 372.688,Z 659.594,A -85,B 0,C 180,E1 -12570.166,E2 -12570.166} C_VEL
LIN {X 0,Y 372.058,Z 671.47,A -85,B 0,C 180,E1 -12571.051,E2 -12571.051} C_VEL
LIN {X 0,Y 371.283,Z 682.176,A -85,B 0,C 180,E1 -12572.064,E2 -12572.064} C_VEL
LIN {X 0,Y 370.491,Z 692.416,A -85,B 0,C 180,E1 -12573.264,E2 -12573.264} C_VEL
LIN {X 0,Y 369.776,Z 702.268,A -85,B 0,C 180,E1 -12574.683,E2 -12574.683} C_VEL
LIN {X 0,Y 369.18,Z 710.464,A -85,B 0,C 180,E1 -12576.143,E2 -12576.143} C_VEL
LIN {X 0,Y 368.553,Z 718.339,A -85,B 0,C 180,E1 -12577.876,E2 -12577.876} C_VEL
LIN {X 0,Y 368.199,Z 723.463,A -85,B 0,C 180,E1 -12579.278,E2 -12579.278} C_VEL
LIN {X 0,Y 367.846,Z 728.626,A -85,B 0,C 180,E1 -12581.047,E2 -12581.047} C_VEL
LIN {X 0,Y 367.647,Z 732.582,A -85,B 0,C 180,E1 -12582.907,E2 -12582.907} C_VEL
LIN {X 0,Y 367.452,Z 734.905,A -85,B 0,C 180,E1 -12584.469,E2 -12584.469} C_VEL
LIN {X 0,Y 367.425,Z 736.017,A -85,B 0,C 180,E1 -12585.602,E2 -12585.602} C_VEL
LIN {X 0,Y 367.498,Z 736.835,A -85,B 0,C 180,E1 -12587.25,E2 -12587.25} C_VEL
LIN {X 0,Y 367.559,Z 736.672,A -85,B 0,C 180,E1 -12588.977,E2 -12588.977} C_VEL
LIN {X 0,Y 367.654,Z 736.027,A -85,B 0,C 180,E1 -12590.094,E2 -12590.094} C_VEL
LIN {X 0,Y 367.814,Z 734.907,A -85,B 0,C 180,E1 -12591.208,E2 -12591.208} C_VEL
LIN {X 0,Y 368.175,Z 732.087,A -85,B 0,C 180,E1 -12593.043,E2 -12593.043} C_VEL
LIN {X 0,Y 368.641,Z 727.464,A -85,B 0,C 180,E1 -12595.079,E2 -12595.079} C_VEL
LIN {X 0,Y 369.226,Z 722.354,A -85,B 0,C 180,E1 -12596.727,E2 -12596.727} C_VEL
LIN {X 0,Y 370.123,Z 714.714,A -85,B 0,C 180,E1 -12598.64,E2 -12598.64} C_VEL
LIN {X 0,Y 371.177,Z 706.39,A -85,B 0,C 180,E1 -12600.272,E2 -12600.272} C_VEL
LIN {X 0,Y 372.141,Z 697.896,A -85,B 0,C 180,E1 -12601.624,E2 -12601.624} C_VEL
LIN {X 0,Y 373.209,Z 687.744,A -85,B 0,C 180,E1 -12602.942,E2 -12602.942} C_VEL
LIN {X 0,Y 374.291,Z 676.684,A -85,B 0,C 180,E1 -12604.081,E2 -12604.081} C_VEL
LIN {X 0,Y 375.135,Z 665.907,A -85,B 0,C 180,E1 -12604.971,E2 -12604.971} C_VEL
LIN {X 0,Y 376.036,Z 653.334,A -85,B 0,C 180,E1 -12605.766,E2 -12605.766} C_VEL
LIN {X 0,Y 376.688,Z 639.5,A -85,B 0,C 180,E1 -12606.394,E2 -12606.394} C_VEL
LIN {X 0,Y 377.247,Z 622.999,A -85,B 0,C 180,E1 -12606.855,E2 -12606.855} C_VEL
LIN {X 0,Y 379.93,Z 545.599,A -85,B 0,C 180,E1 -12608.805,E2 -12608.805} C_VEL
LIN {X 0,Y 376.626,Z 530.154,A -85,B 0,C 180,E1 -12609.562,E2 -12609.562} C_VEL
LIN {X 0,Y 375.845,Z 526.549,A -85,B 0,C 180,E1 -12609.791,E2 -12609.791} C_VEL
LIN {X 0,Y 376.974,Z 507.942,A -85,B 0,C 180,E1 -12613.126,E2 -12613.126} C_VEL
LIN {X 0,Y 375.334,Z 499.408,A -85,B 0,C 180,E1 -12614.92,E2 -12614.92} C_VEL
LIN {X 0,Y 373.317,Z 491.551,A -85,B 0,C 180,E1 -12616.684,E2 -12616.684} C_VEL
LIN {X 0,Y 369.896,Z 481.249,A -85,B 0,C 180,E1 -12619.133,E2 -12619.133} C_VEL
LIN {X 0,Y 368.993,Z 478.64,A -85,B 0,C 180,E1 -12619.869,E2 -12619.869} C_VEL
LIN {X 0,Y 368.942,Z 478.528,A -85,B 0,C 180,E1 -12623.882,E2 -12623.882} C_VEL
LIN {X 0,Y 368.972,Z 478.525,A -85,B 0,C 180,E1 -12627.203,E2 -12627.203} C_VEL
LIN {X 0,Y 368.938,Z 478.531,A -85,B 0,C 180,E1 -12630.953,E2 -12630.953} C_VEL
LIN {X 0,Y 368.938,Z 478.53,A -85,B 0,C 180,E1 -12635.001,E2 -12635.001} C_VEL
LIN {X 0,Y 368.916,Z 478.531,A -85,B 0,C 180,E1 -12638.639,E2 -12638.639} C_VEL
LIN {X 0,Y 368.89,Z 478.533,A -85,B 0,C 180,E1 -12642.009,E2 -12642.009} C_VEL
LIN {X 0,Y 368.888,Z 478.536,A -85,B 0,C 180,E1 -12645.175,E2 -12645.175} C_VEL
LIN {X 0,Y 368.891,Z 478.533,A -85,B 0,C 180,E1 -12648.177,E2 -12648.177} C_VEL
LIN {X 0,Y 368.913,Z 478.506,A -85,B 0,C 180,E1 -12651.359,E2 -12651.359} C_VEL
LIN {X 0,Y 368.976,Z 478.722,A -85,B 0,C 180,E1 -12653.987,E2 -12653.987} C_VEL
LIN {X 0,Y 372.24,Z 491.052,A -85,B 0,C 180,E1 -12656.801,E2 -12656.801} C_VEL
LIN {X 0,Y 375.323,Z 504.429,A -85,B 0,C 180,E1 -12659.628,E2 -12659.628} C_VEL
LIN {X 0,Y 375.792,Z 507.775,A -85,B 0,C 180,E1 -12660.289,E2 -12660.289} C_VEL
LIN {X 0,Y 373.711,Z 527.431,A -85,B 0,C 180,E1 -12663.77,E2 -12663.77} C_VEL
LIN {X 0,Y 372.273,Z 542.832,A -85,B 0,C 180,E1 -12666.421,E2 -12666.421} C_VEL
LIN {X 0,Y 373.446,Z 553.369,A -85,B 0,C 180,E1 -12667.129,E2 -12667.129} C_VEL
LIN {X 0,Y 376.025,Z 572.135,A -85,B 0,C 180,E1 -12667.93,E2 -12667.93} C_VEL
LIN {X 0,Y 377.986,Z 598.154,A -85,B 0,C 180,E1 -12668.849,E2 -12668.849} C_VEL
LIN {X 0,Y 377.217,Z 622.765,A -85,B 0,C 180,E1 -12669.445,E2 -12669.445} C_VEL
LIN {X 0,Y 376.492,Z 661.245,A -85,B 0,C 180,E1 -12670.222,E2 -12670.222} C_VEL
LIN {X 0,Y 375.657,Z 674.884,A -85,B 0,C 180,E1 -12670.71,E2 -12670.71} C_VEL
LIN {X 0,Y 374.254,Z 694.541,A -85,B 0,C 180,E1 -12671.665,E2 -12671.665} C_VEL
LIN {X 0,Y 373.286,Z 706.581,A -85,B 0,C 180,E1 -12672.466,E2 -12672.466} C_VEL
LIN {X 0,Y 372.148,Z 719.042,A -85,B 0,C 180,E1 -12673.543,E2 -12673.543} C_VEL
LIN {X 0,Y 371.007,Z 730.205,A -85,B 0,C 180,E1 -12674.775,E2 -12674.775} C_VEL
LIN {X 0,Y 369.885,Z 740.967,A -85,B 0,C 180,E1 -12676.259,E2 -12676.259} C_VEL
LIN {X 0,Y 369.087,Z 750.45,A -85,B 0,C 180,E1 -12677.908,E2 -12677.908} C_VEL
LIN {X 0,Y 368.392,Z 758.108,A -85,B 0,C 180,E1 -12679.556,E2 -12679.556} C_VEL
LIN {X 0,Y 367.96,Z 764.239,A -85,B 0,C 180,E1 -12681.209,E2 -12681.209} C_VEL
LIN {X 0,Y 367.684,Z 769.046,A -85,B 0,C 180,E1 -12682.861,E2 -12682.861} C_VEL
LIN {X 0,Y 367.587,Z 772.699,A -85,B 0,C 180,E1 -12684.513,E2 -12684.513} C_VEL
LIN {X 0,Y 367.603,Z 774.529,A -85,B 0,C 180,E1 -12685.612,E2 -12685.612} C_VEL
LIN {X 0,Y 367.576,Z 775.929,A -85,B 0,C 180,E1 -12686.71,E2 -12686.71} C_VEL
LIN {X 0,Y 367.705,Z 776.884,A -85,B 0,C 180,E1 -12687.807,E2 -12687.807} C_VEL
LIN {X 0,Y 367.693,Z 777.365,A -85,B 0,C 180,E1 -12688.903,E2 -12688.903} C_VEL
LIN {X 0,Y 367.754,Z 777.43,A -85,B 0,C 180,E1 -12689.998,E2 -12689.998} C_VEL
LIN {X 0,Y 367.709,Z 777.057,A -85,B 0,C 180,E1 -12691.093,E2 -12691.093} C_VEL
LIN {X 0,Y 367.731,Z 776.2,A -85,B 0,C 180,E1 -12692.189,E2 -12692.189} C_VEL
LIN {X 0,Y 367.63,Z 774.901,A -85,B 0,C 180,E1 -12693.286,E2 -12693.286} C_VEL
LIN {X 0,Y 367.694,Z 772.088,A -85,B 0,C 180,E1 -12694.932,E2 -12694.932} C_VEL
LIN {X 0,Y 367.643,Z 768.135,A -85,B 0,C 180,E1 -12696.584,E2 -12696.584} C_VEL
LIN {X 0,Y 367.837,Z 762.961,A -85,B 0,C 180,E1 -12698.237,E2 -12698.237} C_VEL
LIN {X 0,Y 368.12,Z 756.342,A -85,B 0,C 180,E1 -12699.892,E2 -12699.892} C_VEL
LIN {X 0,Y 368.626,Z 748.027,A -85,B 0,C 180,E1 -12701.546,E2 -12701.546} C_VEL
LIN {X 0,Y 369.156,Z 739.484,A -85,B 0,C 180,E1 -12702.924,E2 -12702.924} C_VEL
LIN {X 0,Y 369.756,Z 732.308,A -85,B 0,C 180,E1 -12703.887,E2 -12703.887} C_VEL
LIN {X 0,Y 370.459,Z 721.599,A -85,B 0,C 180,E1 -12705.09,E2 -12705.09} C_VEL
LIN {X 0,Y 371.21,Z 710.526,A -85,B 0,C 180,E1 -12706.073,E2 -12706.073} C_VEL
LIN {X 0,Y 372.062,Z 697.674,A -85,B 0,C 180,E1 -12706.952,E2 -12706.952} C_VEL
LIN {X 0,Y 373.452,Z 677.548,A -85,B 0,C 180,E1 -12708.088,E2 -12708.088} C_VEL
LIN {X 0,Y 374.057,Z 664.315,A -85,B 0,C 180,E1 -12708.589,E2 -12708.589} C_VEL
LIN {X 0,Y 374.442,Z 643.3,A -85,B 0,C 180,E1 -12709.04,E2 -12709.04} C_VEL
LIN {X 0,Y 374.902,Z 595.586,A -85,B 0,C 180,E1 -12709.959,E2 -12709.959} C_VEL
LIN {X 0,Y 370.831,Z 554.824,A -85,B 0,C 180,E1 -12710.977,E2 -12710.977} C_VEL
LIN {X 0,Y 370.586,Z 550.005,A -85,B 0,C 180,E1 -12711.21,E2 -12711.21} C_VEL
LIN {X 0,Y 372.163,Z 527.565,A -85,B 0,C 180,E1 -12714.981,E2 -12714.981} C_VEL
LIN {X 0,Y 373.962,Z 506.071,A -85,B 0,C 180,E1 -12718.633,E2 -12718.633} C_VEL
LIN {X 0,Y 373.916,Z 501.313,A -85,B 0,C 180,E1 -12719.473,E2 -12719.473} C_VEL
LIN {X 0,Y 370.611,Z 486.059,A -85,B 0,C 180,E1 -12722.384,E2 -12722.384} C_VEL
LIN {X 0,Y 368.965,Z 478.641,A -85,B 0,C 180,E1 -12723.897,E2 -12723.897} C_VEL
LIN {X 0,Y 368.889,Z 478.532,A -85,B 0,C 180,E1 -12727.562,E2 -12727.562} C_VEL
LIN {X 0,Y 368.876,Z 478.537,A -85,B 0,C 180,E1 -12730.372,E2 -12730.372} C_VEL
LIN {X 0,Y 368.873,Z 478.534,A -85,B 0,C 180,E1 -12733.614,E2 -12733.614} C_VEL
LIN {X 0,Y 368.877,Z 478.534,A -85,B 0,C 180,E1 -12736.694,E2 -12736.694} C_VEL
LIN {X 0,Y 368.897,Z 478.531,A -85,B 0,C 180,E1 -12739.642,E2 -12739.642} C_VEL
LIN {X 0,Y 368.889,Z 478.531,A -85,B 0,C 180,E1 -12743.143,E2 -12743.143} C_VEL
LIN {X 0,Y 368.886,Z 478.536,A -85,B 0,C 180,E1 -12746.46,E2 -12746.46} C_VEL
LIN {X 0,Y 368.918,Z 478.527,A -85,B 0,C 180,E1 -12749.045,E2 -12749.045} C_VEL
LIN {X 0,Y 368.951,Z 478.525,A -85,B 0,C 180,E1 -12752.795,E2 -12752.795} C_VEL
LIN {X 0,Y 368.932,Z 478.529,A -85,B 0,C 180,E1 -12756.112,E2 -12756.112} C_VEL
LIN {X 0,Y 368.924,Z 478.528,A -85,B 0,C 180,E1 -12759.946,E2 -12759.946} C_VEL
LIN {X 0,Y 368.962,Z 478.521,A -85,B 0,C 180,E1 -12763.398,E2 -12763.398} C_VEL
LIN {X 0,Y 369.045,Z 478.514,A -85,B 0,C 180,E1 -12766.789,E2 -12766.789} C_VEL
LIN {X 0,Y 369.054,Z 478.513,A -85,B 0,C 180,E1 -12770.131,E2 -12770.131} C_VEL
LIN {X 0,Y 369.174,Z 478.5,A -85,B 0,C 180,E1 -12772.342,E2 -12772.342} C_VEL
LIN {X 0,Y 369.128,Z 478.508,A -85,B 0,C 180,E1 -12774.537,E2 -12774.537} C_VEL
LIN {X 0,Y 369.303,Z 478.48,A -85,B 0,C 180,E1 -12777.818,E2 -12777.818} C_VEL
LIN {X 0,Y 369.444,Z 478.463,A -85,B 0,C 180,E1 -12780,E2 -12780} C_VEL
LIN {X 0,Y 369.304,Z 478.482,A -85,B 0,C 180,E1 -12782.181,E2 -12782.181} C_VEL
LIN {X 0,Y 369.183,Z 478.499,A -85,B 0,C 180,E1 -12786.682,E2 -12786.682} C_VEL
LIN {X 0,Y 369.123,Z 478.507,A -85,B 0,C 180,E1 -12788.761,E2 -12788.761} C_VEL
LIN {X 0,Y 368.991,Z 478.519,A -85,B 0,C 180,E1 -12792.093,E2 -12792.093} C_VEL
LIN {X 0,Y 368.984,Z 478.519,A -85,B 0,C 180,E1 -12795.465,E2 -12795.465} C_VEL
LIN {X 0,Y 368.968,Z 478.525,A -85,B 0,C 180,E1 -12798.893,E2 -12798.893} C_VEL
LIN {X 0,Y 368.918,Z 478.53,A -85,B 0,C 180,E1 -12802.396,E2 -12802.396} C_VEL
LIN {X 0,Y 368.986,Z 478.519,A -85,B 0,C 180,E1 -12805.981,E2 -12805.981} C_VEL
LIN {X 0,Y 368.948,Z 478.53,A -85,B 0,C 180,E1 -12808.812,E2 -12808.812} C_VEL
LIN {X 0,Y 368.885,Z 478.533,A -85,B 0,C 180,E1 -12812.239,E2 -12812.239} C_VEL
LIN {X 0,Y 368.916,Z 478.532,A -85,B 0,C 180,E1 -12815.002,E2 -12815.002} C_VEL
LIN {X 0,Y 368.897,Z 478.534,A -85,B 0,C 180,E1 -12818.642,E2 -12818.642} C_VEL
LIN {X 0,Y 368.869,Z 478.533,A -85,B 0,C 180,E1 -12822.011,E2 -12822.011} C_VEL
LIN {X 0,Y 368.944,Z 478.527,A -85,B 0,C 180,E1 -12825.189,E2 -12825.189} C_VEL
LIN {X 0,Y 368.93,Z 478.526,A -85,B 0,C 180,E1 -12828.187,E2 -12828.187} C_VEL
LIN {X 0,Y 368.907,Z 478.531,A -85,B 0,C 180,E1 -12831.359,E2 -12831.359} C_VEL
LIN {X 0,Y 368.927,Z 478.53,A -85,B 0,C 180,E1 -12835.148,E2 -12835.148} C_VEL
LIN {X 0,Y 368.92,Z 478.533,A -85,B 0,C 180,E1 -12839.048,E2 -12839.048} C_VEL
LIN {X 0,Y 368.968,Z 478.522,A -85,B 0,C 180,E1 -12841.565,E2 -12841.565} C_VEL
LIN {X 0,Y 368.992,Z 478.518,A -85,B 0,C 180,E1 -12844.022,E2 -12844.022} C_VEL
LIN {X 0,Y 368.926,Z 478.527,A -85,B 0,C 180,E1 -12847.607,E2 -12847.607} C_VEL
LIN {X 0,Y 368.952,Z 478.529,A -85,B 0,C 180,E1 -12851.108,E2 -12851.108} C_VEL
LIN {X 0,Y 368.993,Z 478.519,A -85,B 0,C 180,E1 -12854.537,E2 -12854.537} C_VEL
LIN {X 0,Y 369.001,Z 478.517,A -85,B 0,C 180,E1 -12857.909,E2 -12857.909} C_VEL
LIN {X 0,Y 369.205,Z 478.496,A -85,B 0,C 180,E1 -12861.825,E2 -12861.825} C_VEL
LIN {X 0,Y 369.238,Z 478.597,A -85,B 0,C 180,E1 -12863.52,E2 -12863.52} C_VEL
LIN {X 0,Y 369.452,Z 479.636,A -85,B 0,C 180,E1 -12863.731,E2 -12863.731} C_VEL
LIN {X 0,Y 375.673,Z 497.161,A -85,B 0,C 180,E1 -12864.393,E2 -12864.393} C_VEL
LIN {X 0,Y 375.095,Z 557.754,A -85,B 0,C 180,E1 -12865.574,E2 -12865.574} C_VEL
LIN {X 0,Y 374.979,Z 571.252,A -85,B 0,C 180,E1 -12866.005,E2 -12866.005} C_VEL
LIN {X 0,Y 374.686,Z 583.899,A -85,B 0,C 180,E1 -12866.641,E2 -12866.641} C_VEL
LIN {X 0,Y 374.248,Z 595.63,A -85,B 0,C 180,E1 -12867.446,E2 -12867.446} C_VEL
LIN {X 0,Y 373.686,Z 606.317,A -85,B 0,C 180,E1 -12868.385,E2 -12868.385} C_VEL
LIN {X 0,Y 372.96,Z 616.875,A -85,B 0,C 180,E1 -12869.545,E2 -12869.545} C_VEL
LIN {X 0,Y 372.272,Z 626.15,A -85,B 0,C 180,E1 -12870.813,E2 -12870.813} C_VEL
LIN {X 0,Y 371.437,Z 635.791,A -85,B 0,C 180,E1 -12872.442,E2 -12872.442} C_VEL
LIN {X 0,Y 370.787,Z 643.501,A -85,B 0,C 180,E1 -12874.078,E2 -12874.078} C_VEL
LIN {X 0,Y 370.147,Z 650.585,A -85,B 0,C 180,E1 -12875.996,E2 -12875.996} C_VEL
LIN {X 0,Y 369.745,Z 655.318,A -85,B 0,C 180,E1 -12877.648,E2 -12877.648} C_VEL
LIN {X 0,Y 369.393,Z 658.964,A -85,B 0,C 180,E1 -12879.308,E2 -12879.308} C_VEL
LIN {X 0,Y 369.158,Z 661.597,A -85,B 0,C 180,E1 -12880.977,E2 -12880.977} C_VEL
LIN {X 0,Y 369.051,Z 662.847,A -85,B 0,C 180,E1 -12882.093,E2 -12882.093} C_VEL
LIN {X 0,Y 369.079,Z 663.914,A -85,B 0,C 180,E1 -12883.8,E2 -12883.8} C_VEL
LIN {X 0,Y 369.174,Z 664.045,A -85,B 0,C 180,E1 -12885.459,E2 -12885.459} C_VEL
LIN {X 0,Y 369.311,Z 663.641,A -85,B 0,C 180,E1 -12886.588,E2 -12886.588} C_VEL
LIN {X 0,Y 369.572,Z 662.477,A -85,B 0,C 180,E1 -12888.043,E2 -12888.043} C_VEL
LIN {X 0,Y 370.076,Z 659.839,A -85,B 0,C 180,E1 -12889.99,E2 -12889.99} C_VEL
LIN {X 0,Y 370.706,Z 656.305,A -85,B 0,C 180,E1 -12891.727,E2 -12891.727} C_VEL
LIN {X 0,Y 371.439,Z 651.715,A -85,B 0,C 180,E1 -12893.414,E2 -12893.414} C_VEL
LIN {X 0,Y 372.445,Z 645.136,A -85,B 0,C 180,E1 -12895.273,E2 -12895.273} C_VEL
LIN {X 0,Y 372.607,Z 643.749,A -85,B 0,C 180,E1 -12895.614,E2 -12895.614} C_VEL
LIN {X 0,Y 372.396,Z 640.626,A -85,B 0,C 180,E1 -12896.386,E2 -12896.386} C_VEL
LIN {X 0,Y 370.482,Z 635.354,A -85,B 0,C 180,E1 -12897.649,E2 -12897.649} C_VEL
LIN {X 0,Y 368.628,Z 629.477,A -85,B 0,C 180,E1 -12898.85,E2 -12898.85} C_VEL
LIN {X 0,Y 368.499,Z 625.41,A -85,B 0,C 180,E1 -12899.514,E2 -12899.514} C_VEL
LIN {X 0,Y 369.496,Z 616.111,A -85,B 0,C 180,E1 -12900.744,E2 -12900.744} C_VEL
LIN {X 0,Y 370.649,Z 604.984,A -85,B 0,C 180,E1 -12901.919,E2 -12901.919} C_VEL
LIN {X 0,Y 371.449,Z 593.446,A -85,B 0,C 180,E1 -12902.875,E2 -12902.875} C_VEL
LIN {X 0,Y 372,Z 581.173,A -85,B 0,C 180,E1 -12903.65,E2 -12903.65} C_VEL
LIN {X 0,Y 372.277,Z 568.443,A -85,B 0,C 180,E1 -12904.223,E2 -12904.223} C_VEL
LIN {X 0,Y 372.374,Z 553.235,A -85,B 0,C 180,E1 -12904.621,E2 -12904.621} C_VEL
LIN {X 0,Y 373.165,Z 503.66,A -85,B 0,C 180,E1 -12905.612,E2 -12905.612} C_VEL
LIN {X 0,Y 364.835,Z 485.867,A -85,B 0,C 180,E1 -12906.654,E2 -12906.654} C_VEL
LIN {X 0,Y 362.03,Z 480.311,A -85,B 0,C 180,E1 -12907.04,E2 -12907.04} C_VEL
LIN {X 0,Y 361.88,Z 479.472,A -85,B 0,C 180,E1 -12907.287,E2 -12907.287} C_VEL
LIN {X 0,Y 361.84,Z 479.413,A -85,B 0,C 180,E1 -12910.757,E2 -12910.757} C_VEL
LIN {X 0,Y 361.822,Z 479.417,A -85,B 0,C 180,E1 -12914.37,E2 -12914.37} C_VEL
LIN {X 0,Y 361.909,Z 479.604,A -85,B 0,C 180,E1 -12917.558,E2 -12917.558} C_VEL
LIN {X 0,Y 365.456,Z 495.368,A -85,B 0,C 180,E1 -12920.736,E2 -12920.736} C_VEL
LIN {X 0,Y 366.628,Z 502.738,A -85,B 0,C 180,E1 -12922.164,E2 -12922.164} C_VEL
LIN {X 0,Y 365.581,Z 523.277,A -85,B 0,C 180,E1 -12925.849,E2 -12925.849} C_VEL
LIN {X 0,Y 366.956,Z 532.598,A -85,B 0,C 180,E1 -12926.188,E2 -12926.188} C_VEL
LIN {X 0,Y 368.954,Z 545.318,A -85,B 0,C 180,E1 -12926.593,E2 -12926.593} C_VEL
LIN {X 0,Y 366.842,Z 633.891,A -85,B 0,C 180,E1 -12928.691,E2 -12928.691} C_VEL
LIN {X 0,Y 366.371,Z 647.389,A -85,B 0,C 180,E1 -12929.225,E2 -12929.225} C_VEL
LIN {X 0,Y 365.729,Z 660.152,A -85,B 0,C 180,E1 -12929.961,E2 -12929.961} C_VEL
LIN {X 0,Y 365.041,Z 672.566,A -85,B 0,C 180,E1 -12930.914,E2 -12930.914} C_VEL
LIN {X 0,Y 364.157,Z 684.472,A -85,B 0,C 180,E1 -12932.095,E2 -12932.095} C_VEL
LIN {X 0,Y 363.377,Z 694.495,A -85,B 0,C 180,E1 -12933.331,E2 -12933.331} C_VEL
LIN {X 0,Y 362.645,Z 703.897,A -85,B 0,C 180,E1 -12934.764,E2 -12934.764} C_VEL
LIN {X 0,Y 362.025,Z 711.865,A -85,B 0,C 180,E1 -12936.246,E2 -12936.246} C_VEL
LIN {X 0,Y 361.439,Z 719.573,A -85,B 0,C 180,E1 -12938.019,E2 -12938.019} C_VEL
LIN {X 0,Y 361.068,Z 724.699,A -85,B 0,C 180,E1 -12939.491,E2 -12939.491} C_VEL
LIN {X 0,Y 360.727,Z 729.523,A -85,B 0,C 180,E1 -12941.249,E2 -12941.249} C_VEL
LIN {X 0,Y 360.555,Z 733.1,A -85,B 0,C 180,E1 -12943,E2 -12943} C_VEL
LIN {X 0,Y 360.391,Z 734.861,A -85,B 0,C 180,E1 -12944.157,E2 -12944.157} C_VEL
LIN {X 0,Y 360.336,Z 736.141,A -85,B 0,C 180,E1 -12945.313,E2 -12945.313} C_VEL
LIN {X 0,Y 360.407,Z 737.215,A -85,B 0,C 180,E1 -12947.169,E2 -12947.169} C_VEL
LIN {X 0,Y 360.467,Z 737.228,A -85,B 0,C 180,E1 -12948.757,E2 -12948.757} C_VEL
LIN {X 0,Y 360.546,Z 736.688,A -85,B 0,C 180,E1 -12949.897,E2 -12949.897} C_VEL
LIN {X 0,Y 360.709,Z 735.732,A -85,B 0,C 180,E1 -12951.033,E2 -12951.033} C_VEL
LIN {X 0,Y 361.116,Z 732.95,A -85,B 0,C 180,E1 -12953.016,E2 -12953.016} C_VEL
LIN {X 0,Y 361.583,Z 728.763,A -85,B 0,C 180,E1 -12954.983,E2 -12954.983} C_VEL
LIN {X 0,Y 362.167,Z 723.949,A -85,B 0,C 180,E1 -12956.663,E2 -12956.663} C_VEL
LIN {X 0,Y 362.944,Z 717.847,A -85,B 0,C 180,E1 -12958.336,E2 -12958.336} C_VEL
LIN {X 0,Y 363.972,Z 710.16,A -85,B 0,C 180,E1 -12960,E2 -12960} C_VEL
LIN {X 0,Y 365.145,Z 700.631,A -85,B 0,C 180,E1 -12961.655,E2 -12961.655} C_VEL
LIN {X 0,Y 366.304,Z 690.888,A -85,B 0,C 180,E1 -12962.997,E2 -12962.997} C_VEL
LIN {X 0,Y 367.498,Z 679.649,A -85,B 0,C 180,E1 -12964.253,E2 -12964.253} C_VEL
LIN {X 0,Y 368.426,Z 669.041,A -85,B 0,C 180,E1 -12965.199,E2 -12965.199} C_VEL
LIN {X 0,Y 369.439,Z 656.249,A -85,B 0,C 180,E1 -12966.075,E2 -12966.075} C_VEL
LIN {X 0,Y 370.114,Z 643.647,A -85,B 0,C 180,E1 -12966.714,E2 -12966.714} C_VEL
LIN {X 0,Y 370.677,Z 629.291,A -85,B 0,C 180,E1 -12967.182,E2 -12967.182} C_VEL
LIN {X 0,Y 373.824,Z 547.839,A -85,B 0,C 180,E1 -12969.281,E2 -12969.281} C_VEL
LIN {X 0,Y 371.85,Z 537.212,A -85,B 0,C 180,E1 -12969.794,E2 -12969.794} C_VEL
LIN {X 0,Y 369.472,Z 527.135,A -85,B 0,C 180,E1 -12970.373,E2 -12970.373} C_VEL
LIN {X 0,Y 370.564,Z 510.234,A -85,B 0,C 180,E1 -12973.453,E2 -12973.453} C_VEL
LIN {X 0,Y 369.048,Z 502.311,A -85,B 0,C 180,E1 -12975.18,E2 -12975.18} C_VEL
LIN {X 0,Y 366.675,Z 493.21,A -85,B 0,C 180,E1 -12977.282,E2 -12977.282} C_VEL
LIN {X 0,Y 363.194,Z 483.087,A -85,B 0,C 180,E1 -12979.794,E2 -12979.794} C_VEL
LIN {X 0,Y 361.895,Z 479.533,A -85,B 0,C 180,E1 -12980.808,E2 -12980.808} C_VEL
LIN {X 0,Y 361.902,Z 479.406,A -85,B 0,C 180,E1 -12984.113,E2 -12984.113} C_VEL
LIN {X 0,Y 361.95,Z 479.398,A -85,B 0,C 180,E1 -12986.721,E2 -12986.721} C_VEL
LIN {X 0,Y 361.882,Z 479.405,A -85,B 0,C 180,E1 -12990.328,E2 -12990.328} C_VEL
LIN {X 0,Y 361.863,Z 479.407,A -85,B 0,C 180,E1 -12994.28,E2 -12994.28} C_VEL
LIN {X 0,Y 361.872,Z 479.409,A -85,B 0,C 180,E1 -12997.222,E2 -12997.222} C_VEL
LIN {X 0,Y 361.844,Z 479.412,A -85,B 0,C 180,E1 -13000.755,E2 -13000.755} C_VEL
LIN {X 0,Y 361.825,Z 479.412,A -85,B 0,C 180,E1 -13004.368,E2 -13004.368} C_VEL
LIN {X 0,Y 361.844,Z 479.414,A -85,B 0,C 180,E1 -13007.567,E2 -13007.567} C_VEL
LIN {X 0,Y 361.875,Z 479.385,A -85,B 0,C 180,E1 -13010.973,E2 -13010.973} C_VEL
LIN {X 0,Y 361.892,Z 479.533,A -85,B 0,C 180,E1 -13013.418,E2 -13013.418} C_VEL
LIN {X 0,Y 365.054,Z 491.41,A -85,B 0,C 180,E1 -13016.232,E2 -13016.232} C_VEL
LIN {X 0,Y 368.05,Z 503.893,A -85,B 0,C 180,E1 -13018.963,E2 -13018.963} C_VEL
LIN {X 0,Y 368.977,Z 509.029,A -85,B 0,C 180,E1 -13020.025,E2 -13020.025} C_VEL
LIN {X 0,Y 366.858,Z 528.531,A -85,B 0,C 180,E1 -13023.549,E2 -13023.549} C_VEL
LIN {X 0,Y 365.702,Z 540.113,A -85,B 0,C 180,E1 -13025.593,E2 -13025.593} C_VEL
LIN {X 0,Y 367.136,Z 553.387,A -85,B 0,C 180,E1 -13026.539,E2 -13026.539} C_VEL
LIN {X 0,Y 369.791,Z 572.562,A -85,B 0,C 180,E1 -13027.387,E2 -13027.387} C_VEL
LIN {X 0,Y 371.639,Z 597.706,A -85,B 0,C 180,E1 -13028.32,E2 -13028.32} C_VEL
LIN {X 0,Y 370.519,Z 630.501,A -85,B 0,C 180,E1 -13029.165,E2 -13029.165} C_VEL
LIN {X 0,Y 369.942,Z 660.224,A -85,B 0,C 180,E1 -13029.785,E2 -13029.785} C_VEL
LIN {X 0,Y 369.149,Z 673.129,A -85,B 0,C 180,E1 -13030.247,E2 -13030.247} C_VEL
LIN {X 0,Y 368.084,Z 689.719,A -85,B 0,C 180,E1 -13030.985,E2 -13030.985} C_VEL
LIN {X 0,Y 367.083,Z 701.796,A -85,B 0,C 180,E1 -13031.727,E2 -13031.727} C_VEL
LIN {X 0,Y 365.983,Z 713.772,A -85,B 0,C 180,E1 -13032.682,E2 -13032.682} C_VEL
LIN {X 0,Y 364.815,Z 724.615,A -85,B 0,C 180,E1 -13033.778,E2 -13033.778} C_VEL
LIN {X 0,Y 363.644,Z 735.708,A -85,B 0,C 180,E1 -13035.184,E2 -13035.184} C_VEL
LIN {X 0,Y 362.671,Z 744.472,A -85,B 0,C 180,E1 -13036.551,E2 -13036.551} C_VEL
LIN {X 0,Y 361.793,Z 753.138,A -85,B 0,C 180,E1 -13038.229,E2 -13038.229} C_VEL
LIN {X 0,Y 361.177,Z 760.155,A -85,B 0,C 180,E1 -13039.912,E2 -13039.912} C_VEL
LIN {X 0,Y 360.789,Z 765.785,A -85,B 0,C 180,E1 -13041.597,E2 -13041.597} C_VEL
LIN {X 0,Y 360.574,Z 770.159,A -85,B 0,C 180,E1 -13043.282,E2 -13043.282} C_VEL
LIN {X 0,Y 360.498,Z 772.42,A -85,B 0,C 180,E1 -13044.404,E2 -13044.404} C_VEL
LIN {X 0,Y 360.526,Z 774.228,A -85,B 0,C 180,E1 -13045.526,E2 -13045.526} C_VEL
LIN {X 0,Y 360.485,Z 775.605,A -85,B 0,C 180,E1 -13046.645,E2 -13046.645} C_VEL
LIN {X 0,Y 360.602,Z 776.507,A -85,B 0,C 180,E1 -13047.764,E2 -13047.764} C_VEL
LIN {X 0,Y 360.623,Z 776.966,A -85,B 0,C 180,E1 -13048.881,E2 -13048.881} C_VEL
LIN {X 0,Y 360.678,Z 777.007,A -85,B 0,C 180,E1 -13049.998,E2 -13049.998} C_VEL
LIN {X 0,Y 360.638,Z 776.589,A -85,B 0,C 180,E1 -13051.115,E2 -13051.115} C_VEL
LIN {X 0,Y 360.663,Z 775.705,A -85,B 0,C 180,E1 -13052.232,E2 -13052.232} C_VEL
LIN {X 0,Y 360.538,Z 774.378,A -85,B 0,C 180,E1 -13053.351,E2 -13053.351} C_VEL
LIN {X 0,Y 360.622,Z 771.507,A -85,B 0,C 180,E1 -13055.029,E2 -13055.029} C_VEL
LIN {X 0,Y 360.573,Z 767.487,A -85,B 0,C 180,E1 -13056.714,E2 -13056.714} C_VEL
LIN {X 0,Y 360.803,Z 761.186,A -85,B 0,C 180,E1 -13058.681,E2 -13058.681} C_VEL
LIN {X 0,Y 361.123,Z 754.222,A -85,B 0,C 180,E1 -13060.369,E2 -13060.369} C_VEL
LIN {X 0,Y 361.617,Z 747.079,A -85,B 0,C 180,E1 -13061.773,E2 -13061.773} C_VEL
LIN {X 0,Y 362.218,Z 738.401,A -85,B 0,C 180,E1 -13063.176,E2 -13063.176} C_VEL
LIN {X 0,Y 362.696,Z 732.031,A -85,B 0,C 180,E1 -13064.041,E2 -13064.041} C_VEL
LIN {X 0,Y 363.469,Z 721.287,A -85,B 0,C 180,E1 -13065.273,E2 -13065.273} C_VEL
LIN {X 0,Y 364.217,Z 710.584,A -85,B 0,C 180,E1 -13066.246,E2 -13066.246} C_VEL
LIN {X 0,Y 365.088,Z 697.854,A -85,B 0,C 180,E1 -13067.142,E2 -13067.142} C_VEL
LIN {X 0,Y 366.504,Z 678.035,A -85,B 0,C 180,E1 -13068.299,E2 -13068.299} C_VEL
LIN {X 0,Y 367.101,Z 665.776,A -85,B 0,C 180,E1 -13068.81,E2 -13068.81} C_VEL
LIN {X 0,Y 367.465,Z 651.823,A -85,B 0,C 180,E1 -13069.158,E2 -13069.158} C_VEL
LIN {X 0,Y 368.151,Z 596.961,A -85,B 0,C 180,E1 -13070.226,E2 -13070.226} C_VEL
LIN {X 0,Y 363.928,Z 554.285,A -85,B 0,C 180,E1 -13071.312,E2 -13071.312} C_VEL
LIN {X 0,Y 363.652,Z 549.26,A -85,B 0,C 180,E1 -13071.541,E2 -13071.541} C_VEL
LIN {X 0,Y 365.317,Z 526.665,A -85,B 0,C 180,E1 -13075.399,E2 -13075.399} C_VEL
LIN {X 0,Y 367.061,Z 506.434,A -85,B 0,C 180,E1 -13078.909,E2 -13078.909} C_VEL
LIN {X 0,Y 367.009,Z 502.904,A -85,B 0,C 180,E1 -13079.542,E2 -13079.542} C_VEL
LIN {X 0,Y 364.018,Z 488.977,A -85,B 0,C 180,E1 -13082.25,E2 -13082.25} C_VEL
LIN {X 0,Y 361.917,Z 479.505,A -85,B 0,C 180,E1 -13084.217,E2 -13084.217} C_VEL
LIN {X 0,Y 361.852,Z 479.407,A -85,B 0,C 180,E1 -13087.22,E2 -13087.22} C_VEL
LIN {X 0,Y 361.804,Z 479.415,A -85,B 0,C 180,E1 -13090.749,E2 -13090.749} C_VEL
LIN {X 0,Y 361.808,Z 479.418,A -85,B 0,C 180,E1 -13094.367,E2 -13094.367} C_VEL
LIN {X 0,Y 361.822,Z 479.412,A -85,B 0,C 180,E1 -13097.567,E2 -13097.567} C_VEL
LIN {X 0,Y 361.818,Z 479.412,A -85,B 0,C 180,E1 -13100.98,E2 -13100.98} C_VEL
LIN {X 0,Y 361.864,Z 479.409,A -85,B 0,C 180,E1 -13104.654,E2 -13104.654} C_VEL
LIN {X 0,Y 361.827,Z 479.417,A -85,B 0,C 180,E1 -13108.369,E2 -13108.369} C_VEL
LIN {X 0,Y 361.896,Z 479.407,A -85,B 0,C 180,E1 -13112.22,E2 -13112.22} C_VEL
LIN {X 0,Y 361.915,Z 479.402,A -85,B 0,C 180,E1 -13114.709,E2 -13114.709} C_VEL
LIN {X 0,Y 361.879,Z 479.41,A -85,B 0,C 180,E1 -13118.346,E2 -13118.346} C_VEL
LIN {X 0,Y 361.955,Z 479.397,A -85,B 0,C 180,E1 -13122.06,E2 -13122.06} C_VEL
LIN {X 0,Y 361.985,Z 479.394,A -85,B 0,C 180,E1 -13126.1,E2 -13126.1} C_VEL
LIN {X 0,Y 362.018,Z 479.388,A -85,B 0,C 180,E1 -13129.937,E2 -13129.937} C_VEL
LIN {X 0,Y 362.137,Z 479.375,A -85,B 0,C 180,E1 -13132.192,E2 -13132.192} C_VEL
LIN {X 0,Y 362.102,Z 479.382,A -85,B 0,C 180,E1 -13134.431,E2 -13134.431} C_VEL
LIN {X 0,Y 362.267,Z 479.356,A -85,B 0,C 180,E1 -13137.776,E2 -13137.776} C_VEL
LIN {X 0,Y 362.413,Z 479.339,A -85,B 0,C 180,E1 -13140,E2 -13140} C_VEL
LIN {X 0,Y 362.268,Z 479.358,A -85,B 0,C 180,E1 -13142.223,E2 -13142.223} C_VEL
LIN {X 0,Y 362.156,Z 479.375,A -85,B 0,C 180,E1 -13146.686,E2 -13146.686} C_VEL
LIN {X 0,Y 362.06,Z 479.385,A -85,B 0,C 180,E1 -13148.933,E2 -13148.933} C_VEL
LIN {X 0,Y 361.947,Z 479.399,A -85,B 0,C 180,E1 -13152.332,E2 -13152.332} C_VEL
LIN {X 0,Y 361.948,Z 479.402,A -85,B 0,C 180,E1 -13154.621,E2 -13154.621} C_VEL
LIN {X 0,Y 361.945,Z 479.397,A -85,B 0,C 180,E1 -13158.1,E2 -13158.1} C_VEL
LIN {X 0,Y 361.878,Z 479.404,A -85,B 0,C 180,E1 -13161.653,E2 -13161.653} C_VEL
LIN {X 0,Y 361.914,Z 479.401,A -85,B 0,C 180,E1 -13165.291,E2 -13165.291} C_VEL
LIN {X 0,Y 361.905,Z 479.401,A -85,B 0,C 180,E1 -13167.779,E2 -13167.779} C_VEL
LIN {X 0,Y 361.833,Z 479.411,A -85,B 0,C 180,E1 -13171.286,E2 -13171.286} C_VEL
LIN {X 0,Y 361.841,Z 479.41,A -85,B 0,C 180,E1 -13174.281,E2 -13174.281} C_VEL
LIN {X 0,Y 361.852,Z 479.41,A -85,B 0,C 180,E1 -13177.224,E2 -13177.224} C_VEL
LIN {X 0,Y 361.824,Z 479.416,A -85,B 0,C 180,E1 -13180.757,E2 -13180.757} C_VEL
LIN {X 0,Y 361.836,Z 479.411,A -85,B 0,C 180,E1 -13184.365,E2 -13184.365} C_VEL
LIN {X 0,Y 361.873,Z 479.405,A -85,B 0,C 180,E1 -13187.561,E2 -13187.561} C_VEL
LIN {X 0,Y 361.868,Z 479.412,A -85,B 0,C 180,E1 -13190.973,E2 -13190.973} C_VEL
LIN {X 0,Y 361.865,Z 479.409,A -85,B 0,C 180,E1 -13194.657,E2 -13194.657} C_VEL
LIN {X 0,Y 361.828,Z 479.411,A -85,B 0,C 180,E1 -13198.372,E2 -13198.372} C_VEL
LIN {X 0,Y 361.892,Z 479.409,A -85,B 0,C 180,E1 -13200.957,E2 -13200.957} C_VEL
LIN {X 0,Y 361.946,Z 479.398,A -85,B 0,C 180,E1 -13203.477,E2 -13203.477} C_VEL
LIN {X 0,Y 361.884,Z 479.409,A -85,B 0,C 180,E1 -13207.147,E2 -13207.147} C_VEL
LIN {X 0,Y 361.901,Z 479.404,A -85,B 0,C 180,E1 -13210.725,E2 -13210.725} C_VEL
LIN {X 0,Y 361.928,Z 479.404,A -85,B 0,C 180,E1 -13213.068,E2 -13213.068} C_VEL
LIN {X 0,Y 361.994,Z 479.391,A -85,B 0,C 180,E1 -13216.53,E2 -13216.53} C_VEL
LIN {X 0,Y 362.028,Z 479.39,A -85,B 0,C 180,E1 -13219.94,E2 -13219.94} C_VEL
LIN {X 0,Y 362.166,Z 479.437,A -85,B 0,C 180,E1 -13223.141,E2 -13223.141} C_VEL
LIN {X 0,Y 362.319,Z 480.258,A -85,B 0,C 180,E1 -13223.366,E2 -13223.366} C_VEL
LIN {X 0,Y 368.873,Z 498.628,A -85,B 0,C 180,E1 -13224.096,E2 -13224.096} C_VEL
LIN {X 0,Y 368.288,Z 558.244,A -85,B 0,C 180,E1 -13225.278,E2 -13225.278} C_VEL
LIN {X 0,Y 368.165,Z 571.254,A -85,B 0,C 180,E1 -13225.691,E2 -13225.691} C_VEL
LIN {X 0,Y 367.903,Z 583.695,A -85,B 0,C 180,E1 -13226.305,E2 -13226.305} C_VEL
LIN {X 0,Y 367.439,Z 595.681,A -85,B 0,C 180,E1 -13227.124,E2 -13227.124} C_VEL
LIN {X 0,Y 366.774,Z 607.945,A -85,B 0,C 180,E1 -13228.218,E2 -13228.218} C_VEL
LIN {X 0,Y 366.063,Z 617.805,A -85,B 0,C 180,E1 -13229.329,E2 -13229.329} C_VEL
LIN {X 0,Y 365.283,Z 628.015,A -85,B 0,C 180,E1 -13230.766,E2 -13230.766} C_VEL
LIN {X 0,Y 364.518,Z 636.373,A -85,B 0,C 180,E1 -13232.212,E2 -13232.212} C_VEL
LIN {X 0,Y 363.84,Z 644.177,A -85,B 0,C 180,E1 -13233.878,E2 -13233.878} C_VEL
LIN {X 0,Y 363.24,Z 650.423,A -85,B 0,C 180,E1 -13235.553,E2 -13235.553} C_VEL
LIN {X 0,Y 362.821,Z 655.391,A -85,B 0,C 180,E1 -13237.235,E2 -13237.235} C_VEL
LIN {X 0,Y 362.426,Z 659.263,A -85,B 0,C 180,E1 -13238.926,E2 -13238.926} C_VEL
LIN {X 0,Y 362.251,Z 661.263,A -85,B 0,C 180,E1 -13240.058,E2 -13240.058} C_VEL
LIN {X 0,Y 362.11,Z 662.856,A -85,B 0,C 180,E1 -13241.193,E2 -13241.193} C_VEL
LIN {X 0,Y 362.015,Z 663.999,A -85,B 0,C 180,E1 -13242.332,E2 -13242.332} C_VEL
LIN {X 0,Y 362.075,Z 664.932,A -85,B 0,C 180,E1 -13243.949,E2 -13243.949} C_VEL
LIN {X 0,Y 362.204,Z 665.001,A -85,B 0,C 180,E1 -13245.764,E2 -13245.764} C_VEL
LIN {X 0,Y 362.335,Z 664.494,A -85,B 0,C 180,E1 -13246.916,E2 -13246.916} C_VEL
LIN {X 0,Y 362.594,Z 663.421,A -85,B 0,C 180,E1 -13248.243,E2 -13248.243} C_VEL
LIN {X 0,Y 362.841,Z 662.262,A -85,B 0,C 180,E1 -13249.227,E2 -13249.227} C_VEL
LIN {X 0,Y 363.399,Z 659.395,A -85,B 0,C 180,E1 -13250.966,E2 -13250.966} C_VEL
LIN {X 0,Y 364.115,Z 655.412,A -85,B 0,C 180,E1 -13252.71,E2 -13252.71} C_VEL
LIN {X 0,Y 365.159,Z 649.135,A -85,B 0,C 180,E1 -13254.749,E2 -13254.749} C_VEL
LIN {X 0,Y 366.246,Z 642.182,A -85,B 0,C 180,E1 -13256.499,E2 -13256.499} C_VEL
LIN {X 0,Y 367.205,Z 635.351,A -85,B 0,C 180,E1 -13257.887,E2 -13257.887} C_VEL
LIN {X 0,Y 368.43,Z 626.045,A -85,B 0,C 180,E1 -13259.421,E2 -13259.421} C_VEL
LIN {X 0,Y 368.499,Z 625.41,A -85,B 0,C 180,E1 -13259.514,E2 -13259.514} C_VEL
LIN {X 0,Y 368.362,Z 621.176,A -85,B 0,C 180,E1 -13260.155,E2 -13260.155} C_VEL
LIN {X 0,Y 366.497,Z 614.212,A -85,B 0,C 180,E1 -13261.222,E2 -13261.222} C_VEL
LIN {X 0,Y 364.621,Z 606.803,A -85,B 0,C 180,E1 -13262.205,E2 -13262.205} C_VEL
LIN {X 0,Y 364.443,Z 601.847,A -85,B 0,C 180,E1 -13262.703,E2 -13262.703} C_VEL
LIN {X 0,Y 365.2,Z 590.302,A -85,B 0,C 180,E1 -13263.594,E2 -13263.594} C_VEL
LIN {X 0,Y 365.731,Z 577.428,A -85,B 0,C 180,E1 -13264.326,E2 -13264.326} C_VEL
LIN {X 0,Y 365.95,Z 565.221,A -85,B 0,C 180,E1 -13264.804,E2 -13264.804} C_VEL
LIN {X 0,Y 366.2,Z 534.318,A -85,B 0,C 180,E1 -13265.487,E2 -13265.487} C_VEL
LIN {X 0,Y 366.828,Z 505.672,A -85,B 0,C 180,E1 -13266.059,E2 -13266.059} C_VEL
LIN {X 0,Y 359.043,Z 489.255,A -85,B 0,C 180,E1 -13267.06,E2 -13267.06} C_VEL
LIN {X 0,Y 355.033,Z 481.235,A -85,B 0,C 180,E1 -13267.616,E2 -13267.616} C_VEL
LIN {X 0,Y 354.852,Z 480.346,A -85,B 0,C 180,E1 -13267.879,E2 -13267.879} C_VEL
LIN {X 0,Y 354.792,Z 480.292,A -85,B 0,C 180,E1 -13271.173,E2 -13271.173} C_VEL
LIN {X 0,Y 354.768,Z 480.295,A -85,B 0,C 180,E1 -13274.508,E2 -13274.508} C_VEL
LIN {X 0,Y 354.883,Z 480.544,A -85,B 0,C 180,E1 -13277.264,E2 -13277.264} C_VEL
LIN {X 0,Y 358.573,Z 496.953,A -85,B 0,C 180,E1 -13280.598,E2 -13280.598} C_VEL
LIN {X 0,Y 359.731,Z 504.214,A -85,B 0,C 180,E1 -13282.019,E2 -13282.019} C_VEL
LIN {X 0,Y 358.731,Z 523.708,A -85,B 0,C 180,E1 -13285.541,E2 -13285.541} C_VEL
LIN {X 0,Y 361.153,Z 539.757,A -85,B 0,C 180,E1 -13286.109,E2 -13286.109} C_VEL
LIN {X 0,Y 362.142,Z 546.346,A -85,B 0,C 180,E1 -13286.319,E2 -13286.319} C_VEL
LIN {X 0,Y 359.906,Z 634.696,A -85,B 0,C 180,E1 -13288.469,E2 -13288.469} C_VEL
LIN {X 0,Y 359.481,Z 646.926,A -85,B 0,C 180,E1 -13288.96,E2 -13288.96} C_VEL
LIN {X 0,Y 358.801,Z 659.907,A -85,B 0,C 180,E1 -13289.711,E2 -13289.711} C_VEL
LIN {X 0,Y 358.132,Z 671.767,A -85,B 0,C 180,E1 -13290.62,E2 -13290.62} C_VEL
LIN {X 0,Y 357.322,Z 682.593,A -85,B 0,C 180,E1 -13291.673,E2 -13291.673} C_VEL
LIN {X 0,Y 356.449,Z 693.741,A -85,B 0,C 180,E1 -13293.033,E2 -13293.033} C_VEL
LIN {X 0,Y 355.652,Z 703.712,A -85,B 0,C 180,E1 -13294.546,E2 -13294.546} C_VEL
LIN {X 0,Y 355.003,Z 711.786,A -85,B 0,C 180,E1 -13296.057,E2 -13296.057} C_VEL
LIN {X 0,Y 354.386,Z 719.615,A -85,B 0,C 180,E1 -13297.865,E2 -13297.865} C_VEL
LIN {X 0,Y 353.959,Z 725.71,A -85,B 0,C 180,E1 -13299.668,E2 -13299.668} C_VEL
LIN {X 0,Y 353.621,Z 730.404,A -85,B 0,C 180,E1 -13301.459,E2 -13301.459} C_VEL
LIN {X 0,Y 353.524,Z 732.866,A -85,B 0,C 180,E1 -13302.651,E2 -13302.651} C_VEL
LIN {X 0,Y 353.349,Z 734.756,A -85,B 0,C 180,E1 -13303.832,E2 -13303.832} C_VEL
LIN {X 0,Y 353.257,Z 736.193,A -85,B 0,C 180,E1 -13305.011,E2 -13305.011} C_VEL
LIN {X 0,Y 353.335,Z 737.592,A -85,B 0,C 180,E1 -13307.073,E2 -13307.073} C_VEL
LIN {X 0,Y 353.387,Z 737.722,A -85,B 0,C 180,E1 -13308.529,E2 -13308.529} C_VEL
LIN {X 0,Y 353.443,Z 737.349,A -85,B 0,C 180,E1 -13309.691,E2 -13309.691} C_VEL
LIN {X 0,Y 353.621,Z 736.501,A -85,B 0,C 180,E1 -13310.852,E2 -13310.852} C_VEL
LIN {X 0,Y 354.053,Z 733.82,A -85,B 0,C 180,E1 -13312.993,E2 -13312.993} C_VEL
LIN {X 0,Y 354.526,Z 730.096,A -85,B 0,C 180,E1 -13314.882,E2 -13314.882} C_VEL
LIN {X 0,Y 355.113,Z 725.519,A -85,B 0,C 180,E1 -13316.597,E2 -13316.597} C_VEL
LIN {X 0,Y 356.061,Z 718.578,A -85,B 0,C 180,E1 -13318.587,E2 -13318.587} C_VEL
LIN {X 0,Y 357.153,Z 710.954,A -85,B 0,C 180,E1 -13320.282,E2 -13320.282} C_VEL
LIN {X 0,Y 358.412,Z 701.544,A -85,B 0,C 180,E1 -13321.967,E2 -13321.967} C_VEL
LIN {X 0,Y 359.645,Z 691.77,A -85,B 0,C 180,E1 -13323.361,E2 -13323.361} C_VEL
LIN {X 0,Y 360.898,Z 680.898,A -85,B 0,C 180,E1 -13324.608,E2 -13324.608} C_VEL
LIN {X 0,Y 361.877,Z 670.473,A -85,B 0,C 180,E1 -13325.573,E2 -13325.573} C_VEL
LIN {X 0,Y 362.926,Z 657.969,A -85,B 0,C 180,E1 -13326.463,E2 -13326.463} C_VEL
LIN {X 0,Y 363.655,Z 645.171,A -85,B 0,C 180,E1 -13327.147,E2 -13327.147} C_VEL
LIN {X 0,Y 364.266,Z 631.647,A -85,B 0,C 180,E1 -13327.623,E2 -13327.623} C_VEL
LIN {X 0,Y 367.649,Z 547.862,A -85,B 0,C 180,E1 -13329.862,E2 -13329.862} C_VEL
LIN {X 0,Y 364.052,Z 531.252,A -85,B 0,C 180,E1 -13330.772,E2 -13330.772} C_VEL
LIN {X 0,Y 363.175,Z 527.619,A -85,B 0,C 180,E1 -13331.017,E2 -13331.017} C_VEL
LIN {X 0,Y 364.226,Z 513.133,A -85,B 0,C 180,E1 -13333.691,E2 -13333.691} C_VEL
LIN {X 0,Y 362.778,Z 505.228,A -85,B 0,C 180,E1 -13335.449,E2 -13335.449} C_VEL
LIN {X 0,Y 360.477,Z 496.199,A -85,B 0,C 180,E1 -13337.589,E2 -13337.589} C_VEL
LIN {X 0,Y 357.558,Z 487.5,A -85,B 0,C 180,E1 -13339.819,E2 -13339.819} C_VEL
LIN {X 0,Y 354.853,Z 480.442,A -85,B 0,C 180,E1 -13341.847,E2 -13341.847} C_VEL
LIN {X 0,Y 354.907,Z 480.278,A -85,B 0,C 180,E1 -13345.827,E2 -13345.827} C_VEL
LIN {X 0,Y 354.827,Z 480.285,A -85,B 0,C 180,E1 -13349.681,E2 -13349.681} C_VEL
LIN {X 0,Y 354.815,Z 480.285,A -85,B 0,C 180,E1 -13353.701,E2 -13353.701} C_VEL
LIN {X 0,Y 354.806,Z 480.287,A -85,B 0,C 180,E1 -13356.459,E2 -13356.459} C_VEL
LIN {X 0,Y 354.833,Z 480.286,A -85,B 0,C 180,E1 -13359.423,E2 -13359.423} C_VEL
LIN {X 0,Y 354.797,Z 480.289,A -85,B 0,C 180,E1 -13362.866,E2 -13362.866} C_VEL
LIN {X 0,Y 354.775,Z 480.291,A -85,B 0,C 180,E1 -13366.103,E2 -13366.103} C_VEL
LIN {X 0,Y 354.796,Z 480.292,A -85,B 0,C 180,E1 -13369.178,E2 -13369.178} C_VEL
LIN {X 0,Y 354.858,Z 480.387,A -85,B 0,C 180,E1 -13372.837,E2 -13372.837} C_VEL
LIN {X 0,Y 357.877,Z 491.467,A -85,B 0,C 180,E1 -13375.569,E2 -13375.569} C_VEL
LIN {X 0,Y 361.177,Z 505.32,A -85,B 0,C 180,E1 -13378.687,E2 -13378.687} C_VEL
